// ---- POUs/20_AUTO/ST128/FB_AUT_128.TcPOU
FUNCTION_BLOCK FB_AUT_128 EXTENDS FB_AUT_ABSTRACT
(****************************************************************************)
(*	POU_AUT_zxx			Bausteinaufrufe Station	zxx							*)
(*	Status				ungetestet											*)
(*  Version:			1.0													*)
(*	Beschrieb:																*)
(*																			*)
(*	Abläufe:			FB_ABLzxxA		Hauptablauf							*)
(*																			*)
(*																			*)
(* 	25.09.2019/Dj															*)
(****************************************************************************)
(*	dd.mm.yyyy   KZ    x.y			Beschrieb								*)
(****************************************************************************)
VAR_INPUT
    (* spezifische Eingänge *)

END_VAR
VAR_OUTPUT
    (* spezifische Ausgänge *)

END_VAR
VAR
    (* Bausteine *)
    fb_TubeCapCheck : FB_ABL_128_TubeCapCheck; // 

    fb_stat : FB_AUT_Statistics;
END_VAR

(*******************************************************************)
(* Timer *)
(*******************************************************************)

(*******************************************************************)
(* Flanken / Merker *)
(*******************************************************************)
//MANU CYCLE
IF (enIN_State = StateMANU) AND xIN_ManuCycle THEN
    xManuCycle := TRUE;
END_IF;

IF (enIN_State <> StateMANU) OR xOUT_Done THEN
    xManuCycle := FALSE;
END_IF

//NEXT STEP
xNextStep := (enIN_State > StateSTEP) OR
             ((enIN_State = StateSTEP) AND xIN_Step) OR
             ((enIN_State = StateMANU) AND xManuCycle);

//RESET
xReset := (enIN_State < StateREADY) AND (enIN_State <> StateINIT) AND NOT xManuCycle;

(*******************************************************************)
(* Bausteinaufrufe Abläufe *)
(*******************************************************************)

xRelease := MAIN.MoverMan.IsProcessUsed(THIS^);

fb_TubeCapCheck(xIN_Reset       := xReset,
                xIN_Init        := xIN_Init,
                xIN_Quit        := xIN_Quit,
                xIN_Start       := enIN_State >= enState.StateLEER AND xRelease,
                xIN_Sperre      := NOT xIN_On,
                xIN_NextStep    := xNextStep,
                xIN_AlarmAktiv  := xIN_AlarmAktiv,
                xIN_DryCycle    := xIN_DryCycle,
                xIN_RestartCYCL := enIN_State >= enState.StateLEER,
                enIN_State      := enIN_State,
                tIN_Timeout     := tIN_Timeout,
                pxFG_Freigabe   := ADR(xRelease),
                Mover           := THIS^.Mover);

fb_stat(xIN_Enable  := enState.StateAUTO = enIN_State,
        xIN_Waiting := fb_TubeCapCheck.xOUT_Wait,
        xIN_Running := (fb_TubeCapCheck.iOUT_Step >= ST128_TubeCapCheck_e.START) AND
                       (fb_TubeCapCheck.iOUT_Step <= ST128_TubeCapCheck_e.DONE),
        // Since we use a mover system, a cycle is done when we are waiting on a mover
        xIN_Done := fb_TubeCapCheck.iOUT_Step = ST128_TubeCapCheck_e.waitOnMover);

(*******************************************************************)
(* Mover reset flags *)
(*******************************************************************)

(*******************************************************************)
(* OUTPUT *)
(*******************************************************************)
xOUT_InitDone := fb_TubeCapCheck.xOUT_InitDone;
xOUT_Ready    := fb_TubeCapCheck.xOUT_Ready;
xOUT_Done     := fb_TubeCapCheck.xOUT_Done;
xOUT_ErrFlag  := fb_TubeCapCheck.xOUT_ErrFlag;
xOUT_Wait     := fb_TubeCapCheck.xOUT_Wait;
xOUT_AlarmST  := xOUT_ErrFlag;

(*******************************************************************)
(* Bausteinaufruf Error Station *)
(*******************************************************************)
// POU_ERR_VORLAGE(xIN_QUIT:=xIN_Quit , pstrArIN_ALARM:=ADR(HMI.strArALARM[1]));

(* % of completion of the process *)
PROPERTY iCompletionPC : INT
GET
iCompletionPC := THIS^.fb_TubeCapCheck.iOUT_ProcessCompletion;
END_GET
END_PROPERTY

PROPERTY ProcessExecution : ProcessExecution_e
GET
ProcessExecution := THIS^._ProcessExecution;
END_GET
SET
THIS^._ProcessExecution := ProcessExecution;
END_SET
END_PROPERTY

PROPERTY xBusy : BOOL
GET
xBusy := THIS^.fb_TubeCapCheck.xOUT_Busy;
END_GET
SET
END_SET
END_PROPERTY

PROPERTY xDone : BOOL
GET
xDone := THIS^.fb_TubeCapCheck.xOUT_Ready OR THIS^.fb_TubeCapCheck.xOUT_Done;
END_GET
END_PROPERTY

PROPERTY xMoverPathFree : BOOL
GET
xMoverPathFree := THIS^.fb_TubeCapCheck.xOUT_MoverFree OR THIS^.fb_TubeCapCheck.xOUT_Ready OR THIS^.fb_TubeCapCheck.xOUT_Done;
END_GET
END_PROPERTY

PROPERTY xMoverShouldLeave : BOOL
GET
xMoverShouldLeave := THIS^.fb_TubeCapCheck.iOUT_Step = ST128_TubeCapCheck_e.SYNC_MOVER_LEAVE;
END_GET
END_PROPERTY

END_FUNCTION_BLOCK

// ---- POUs/20_AUTO/ST140/FB_AUT_140.TcPOU
FUNCTION_BLOCK FB_AUT_140 EXTENDS FB_AUT_ABSTRACT
(****************************************************************************)
(*	POU_AUT_zxx			Bausteinaufrufe Station	zxx							*)
(*	Status				ungetestet											*)
(*  Version:			1.0													*)
(*	Beschrieb:																*)
(*																			*)
(*	Abläufe:			FB_ABLzxxA		Hauptablauf							*)
(*																			*)
(*																			*)
(* 	25.09.2019/Dj															*)
(****************************************************************************)
(*	dd.mm.yyyy   KZ    x.y			Beschrieb								*)
(****************************************************************************)
VAR_INPUT
    (* spezifische Eingänge *)

END_VAR
VAR_OUTPUT
    (* spezifische Ausgänge *)

END_VAR
VAR
    (* Bausteine *)
    fb_Measure : FB_ABL_140_Measure;

    fb_stat : FB_AUT_Statistics;

END_VAR

(*******************************************************************)
(* Timer *)
(*******************************************************************)

(*******************************************************************)
(* Flanken / Merker *)
(*******************************************************************)
//MANU CYCLE
IF (enIN_State = StateMANU) AND xIN_ManuCycle THEN
    xManuCycle := TRUE;
END_IF;

IF (enIN_State <> StateMANU) OR xOUT_Done THEN
    xManuCycle := FALSE;
END_IF

//NEXT STEP
xNextStep := (enIN_State > StateSTEP) OR
             ((enIN_State = StateSTEP) AND xIN_Step) OR
             ((enIN_State = StateMANU) AND xManuCycle);

//RESET
xReset := (enIN_State < StateREADY) AND (enIN_State <> StateINIT) AND NOT xManuCycle;

(*******************************************************************)
(* Bausteinaufrufe Abläufe *)
(*******************************************************************)

xRelease := MAIN.MoverMan.IsProcessUsed(THIS^);

fb_Measure(xIN_Reset       := xReset,
           xIN_Init        := xIN_Init,
           xIN_Quit        := xIN_Quit,
           xIN_Start       := enIN_State >= enState.StateLEER AND xRelease,
           xIN_Sperre      := NOT xIN_On,
           xIN_NextStep    := xNextStep,
           xIN_AlarmAktiv  := xIN_AlarmAktiv,
           xIN_DryCycle    := xIN_DryCycle,
           xIN_RestartCYCL := enIN_State >= enState.StateLEER,
           enIN_State      := enIN_State,
           tIN_Timeout     := tIN_Timeout,
           pxFG_Freigabe   := ADR(xRelease),
           Mover           := THIS^.Mover);

fb_stat(xIN_Enable  := enState.StateAUTO = enIN_State,
        xIN_Waiting := fb_Measure.xOUT_Wait,
        xIN_Running := (fb_Measure.iOUT_Step >= ST140_Measure_e.START) AND
                       (fb_Measure.iOUT_Step <= ST140_Measure_e.DONE),
        // Since we use a mover system, a cycle is done when we are waiting on a mover
        xIN_Done := fb_Measure.iOUT_Step = ST140_Measure_e.waitOnMover);

(*******************************************************************)
(* Mover reset flags *)
(*******************************************************************)

(*******************************************************************)
(* OUTPUT *)
(*******************************************************************)
xOUT_InitDone := fb_Measure.xOUT_InitDone;
xOUT_Ready    := fb_Measure.xOUT_Ready;
xOUT_Done     := fb_Measure.xOUT_Done;
xOUT_ErrFlag  := fb_Measure.xOUT_ErrFlag;
xOUT_Wait     := fb_Measure.xOUT_Wait;
xOUT_AlarmST  := xOUT_ErrFlag;

(*******************************************************************)
(* Bausteinaufruf Error Station *)
(*******************************************************************)
// POU_ERR_VORLAGE(xIN_QUIT:=xIN_Quit , pstrArIN_ALARM:=ADR(HMI.strArALARM[1]));

(* % of completion of the process *)
PROPERTY iCompletionPC : INT
GET
iCompletionPC := THIS^.fb_Measure.iOUT_ProcessCompletion;
END_GET
END_PROPERTY

PROPERTY ProcessExecution : ProcessExecution_e
GET
ProcessExecution := THIS^._ProcessExecution;
END_GET
SET
THIS^._ProcessExecution := ProcessExecution;
END_SET
END_PROPERTY

PROPERTY xBusy : BOOL
GET
xBusy := THIS^.fb_Measure.xOUT_Busy;
END_GET
SET
END_SET
END_PROPERTY

PROPERTY xDone : BOOL
GET
xDone := THIS^.fb_Measure.xOUT_Ready OR THIS^.fb_Measure.xOUT_Done;
END_GET
END_PROPERTY

PROPERTY xMoverPathFree : BOOL
GET
xMoverPathFree := THIS^.fb_Measure.xOUT_MoverFree OR THIS^.fb_Measure.xOUT_Ready OR THIS^.fb_Measure.xOUT_Done;
END_GET
END_PROPERTY

PROPERTY xMoverShouldLeave : BOOL
GET
xMoverShouldLeave := THIS^.fb_Measure.iOUT_Step = ST140_Measure_e.SYNC_MOVER_LEAVE;
END_GET
END_PROPERTY

END_FUNCTION_BLOCK

// ---- POUs/20_AUTO/ST145/FB_AUT_145.TcPOU
FUNCTION_BLOCK FB_AUT_145 EXTENDS FB_AUT_ABSTRACT
(****************************************************************************)
(*	POU_AUT_zxx			Bausteinaufrufe Station	zxx							*)
(*	Status				ungetestet											*)
(*  Version:			1.0													*)
(*	Beschrieb:																*)
(*																			*)
(*	Abläufe:			FB_ABLzxxA		Hauptablauf							*)
(*																			*)
(*																			*)
(* 	25.09.2019/Dj															*)
(****************************************************************************)
(*	dd.mm.yyyy   KZ    x.y			Beschrieb								*)
(****************************************************************************)
VAR_INPUT
    (* spezifische Eingänge *)

END_VAR
VAR_OUTPUT
    (* spezifische Ausgänge *)

END_VAR
VAR
    (* Bausteine *)
    fb_Pnp    : FB_ABL_145_Pnp;
    fb_Feeder : FB_ABL_145_Feeder;

    fb_stat_pnp    : FB_AUT_Statistics;
    fb_stat_Feeder : FB_AUT_Statistics;

END_VAR

VAR CONSTANT
    ROT_TABLE_FREE_MAX_Y : REAL := 100.0; // If Y and Z axis is more than this value, the feeder cannot move
    ROT_TABLE_FREE_MAX_Z : REAL := 50.0; // If Z and Y axis is more than this value, the feeder cannot move

    PNP_VERTICAL_MAX_Z : REAL := 50.0; // If Z axis is more than this value, the horizontal axis of the pnp cannot move
END_VAR

(*******************************************************************)
(* Timer *)
(*******************************************************************)

(*******************************************************************)
(* Flanken / Merker *)
(*******************************************************************)
//MANU CYCLE
IF (enIN_State = StateMANU) AND xIN_ManuCycle THEN
    xManuCycle := TRUE;
END_IF;

IF (enIN_State <> StateMANU) OR xOUT_Done THEN
    xManuCycle := FALSE;
END_IF

//NEXT STEP
xNextStep := (enIN_State > StateSTEP) OR
             ((enIN_State = StateSTEP) AND xIN_Step) OR
             ((enIN_State = StateMANU) AND xManuCycle);

//RESET
xReset := (enIN_State < StateREADY) AND (enIN_State <> StateINIT) AND NOT xManuCycle;

(*******************************************************************)
(* Bausteinaufrufe Abläufe *)
(*******************************************************************)

xRelease := MAIN.MoverMan.IsProcessUsed(THIS^);

fb_Pnp(xIN_Reset          := xReset,
       xIN_Init           := xIN_Init,
       xIN_Quit           := xIN_Quit,
       xIN_Start          := enIN_State >= enState.StateLEER AND xRelease,
       xIN_Sperre         := NOT xIN_On,
       xIN_NextStep       := xNextStep,
       xIN_AlarmAktiv     := xIN_AlarmAktiv,
       xIN_DryCycle       := xIN_DryCycle,
       xIN_RestartCYCL    := enIN_State >= enState.StateLEER,
       enIN_State         := enIN_State,
       tIN_Timeout        := tIN_Timeout,
       pxFG_Freigabe      := ADR(xRelease),
       Mover              := THIS^.Mover,
       xIN_PceReadyToPick := fb_Feeder.xOUT_Done,
       xIN_HorAxisFree    := ST145_Axis.axis145_02Z.rActPos < ROT_TABLE_FREE_MAX_Y);

fb_Feeder(xIN_Reset       := xReset,
          xIN_Init        := xIN_Init,
          xIN_Quit        := xIN_Quit,
          xIN_Start       := enIN_State >= enState.StateLEER AND xRelease,
          xIN_Sperre      := NOT xIN_On,
          xIN_NextStep    := xNextStep,
          xIN_AlarmAktiv  := xIN_AlarmAktiv,
          xIN_DryCycle    := xIN_DryCycle,
          xIN_RestartCYCL := enIN_State >= enState.StateLEER,
          enIN_State      := enIN_State,
          tIN_Timeout     := tIN_Timeout,
          pxFG_Freigabe   := ADR(xRelease),
          // special
          xIN_PickPiece            := fb_Pnp.xOUT_PickPiece,
          xIN_RotTableBlockedByPnp := (ST145_Axis.axis145_01Y.rActPos > ROT_TABLE_FREE_MAX_Y) AND
                                      (ST145_Axis.axis145_02Z.rActPos > ROT_TABLE_FREE_MAX_Z));

fb_stat_pnp(xIN_Enable  := enState.StateAUTO = enIN_State,
            xIN_Waiting := fb_Pnp.xOUT_Wait,
            xIN_Running := (fb_Pnp.iOUT_Step >= ST145_Pnp_e.START) AND
                           (fb_Pnp.iOUT_Step <= ST145_Pnp_e.DONE),
            // Since we use a mover system, a cycle is done when we are waiting on a mover
            xIN_Done := fb_Pnp.iOUT_Step = ST145_Pnp_e.waitOnMover);

fb_stat_Feeder(xIN_Enable  := enState.StateAUTO = enIN_State,
               xIN_Waiting := fb_feeder.xOUT_Wait,
               xIN_Running := (fb_feeder.iOUT_Step >= ST145_Feeder_e.START) AND
                              (fb_feeder.iOUT_Step <= ST145_Feeder_e.DONE),
               xIN_Done := fb_feeder.iOUT_Step = ST145_Feeder_e.DONE);

(*******************************************************************)
(* Mover reset flags *)
(*******************************************************************)

(*******************************************************************)
(* OUTPUT *)
(*******************************************************************)
xOUT_InitDone := fb_Pnp.xOUT_InitDone AND fb_Feeder.xOUT_InitDone;
xOUT_Ready    := fb_Pnp.xOUT_Ready AND fb_Feeder.xOUT_Ready;
xOUT_Done     := fb_Pnp.xOUT_Done; // we ignore feeder
xOUT_ErrFlag  := fb_Pnp.xOUT_ErrFlag OR fb_Feeder.xOUT_ErrFlag;
xOUT_Wait     := fb_Pnp.xOUT_Wait AND fb_Feeder.xOUT_Wait;
xOUT_AlarmST  := xOUT_ErrFlag;

(*******************************************************************)
(* Bausteinaufruf Error Station *)
(*******************************************************************)
// POU_ERR_VORLAGE(xIN_QUIT:=xIN_Quit , pstrArIN_ALARM:=ADR(HMI.strArALARM[1]));

(* % of completion of the process *)
PROPERTY iCompletionPC : INT
GET
iCompletionPC := THIS^.fb_Pnp.iOUT_ProcessCompletion;
END_GET
END_PROPERTY

PROPERTY ProcessExecution : ProcessExecution_e
GET
ProcessExecution := THIS^._ProcessExecution;
END_GET
SET
THIS^._ProcessExecution := ProcessExecution;
END_SET
END_PROPERTY

PROPERTY xBusy : BOOL
GET
xBusy := THIS^.fb_Pnp.xOUT_Busy;
END_GET
SET
END_SET
END_PROPERTY

PROPERTY xDone : BOOL
GET
xDone := THIS^.fb_Pnp.xOUT_Ready OR THIS^.fb_Pnp.xOUT_Done;
END_GET
END_PROPERTY

PROPERTY xMoverPathFree : BOOL
GET
xMoverPathFree := THIS^.fb_Pnp.xOUT_MoverFree OR THIS^.fb_Pnp.xOUT_Ready OR THIS^.fb_Pnp.xOUT_Done;
END_GET
END_PROPERTY

PROPERTY xMoverShouldLeave : BOOL
GET
xMoverShouldLeave := THIS^.fb_Pnp.iOUT_Step = ST145_Pnp_e.SYNC_MOVER_LEAVE;
END_GET
END_PROPERTY

END_FUNCTION_BLOCK

// ---- POUs/20_AUTO/ST15x/FB_ABL_150.TcPOU
FUNCTION_BLOCK FB_ABL_150
(****************************************************************************************)
(*	TITEL				laden kristall- Modul	    										*)
(*	Status				ungetestet                         								*)
(*	Beschrieb:			Ablaufbeschreibung												*)
(*																						*)
(*	Steps:	self-explained using enum													*)
(***********************************Revisionen*******************************************)
(*	see github blames																	*)
(****************************************************************************************)

VAR_INPUT
    xIN_Reset       : BOOL;          // Schrittkette zurücksetzen 
    xIN_Init        : BOOL;          // Initialisieren
    xIN_Quit        : BOOL;          // Fehler quittieren 
    xIN_Start       : BOOL;          // Startbefehl
    xIN_Sperre      : BOOL;          // FB Sperren 
    xIN_NextStep    : BOOL;          // Nächsten Schritt ausführen 
    xIN_AlarmAktiv  : BOOL;          // Anlage hat Alarm
    xIN_DryCycle    : BOOL;          // Fahren ohne Teile
    xIN_RestartCYCL : BOOL;          // Zyklus erneut starten im STEP, END, LEERFAHREN
    enIN_State      : enState;       // Status Anlage
    tIN_Timeout     : TIME := T#10s; // Timout

    pxFG_Freigabe : POINTER TO BOOL; //Freigabe von Station

    // Application specific
    Mover : REFERENCE TO FB_Mover;

    xIN_capDetector             : BOOL;
    xIN_kraftubersetzunh_zuruck : BOOL;
    xIN_kraftubersetzunh_vor    : BOOL;
    pIN_ButtonMaintaining       : POINTER TO structButton;

    xIN_welding_bits : Ultrasonic_IN_bits_t;

    iIN_StationNumber : INT;    // station number 
    sIN_errorCodeSide : STRING; // added string to the error code, (e.g. left or right)

END_VAR
VAR_OUTPUT
    (* standart Ausgänge *)
    xOUT_ErrFlag  : BOOL;        // Error Flag 
    xOUT_Busy     : BOOL;        // Baustein befindet sich im Ablauf 
    xOUT_Done     : BOOL;        // Baustein hat den Ablauf beendet 		
    xOUT_Ready    : BOOL;        // Ready to begin, should be the same state as done	
    xOUT_Timeout  : BOOL;        // Timeout FB 
    xOUT_InitDone : BOOL;        // initialisierung fertig
    xOUT_Wait     : BOOL;        // Wartet auf Bedingung
    iOUT_Step     : ST150_Uss_e; // Aktueller Schritt 
    sOUT_Step     : STRING;      // Aktueller Schritt but in string format
    bOUT_Error    : BYTE;        // Fehlernummer

    iOUT_ProcessCompletion : INT;  //process completion, express in % (0-100)
    xOUT_MoverFree         : BOOL; // The mover is free to move

    xOUT_moverMaintening_valve : BOOL;
    xOUT_welding_bits          : Ultrasonic_OUT_bits_t;

END_VAR
VAR
    (* Standard *)
    (* Schritt *)
    iLastStep : ST150_Uss_e; // Merker letzter Schritt 
    iPreStep  : ST150_Uss_e; // Schritt zurück nach Alarm 
    iAktStep  : ST150_Uss_e; // aktueller Schritt

    // Trigger Starten 
    rtSTART : R_TRIG;
    // Timer TimeOut 
    TON_Timeout : TON;

    (* Bausteine *)

    (* Spezial *)
    fb_moverMaintening   : FB_ZylMo2El_V2_1;
    simu_moverMaintening : FB_Simu_Zyl2Pos;

    TON_UssError     : TON;
    TON_CapDetection : TON;

END_VAR
VAR CONSTANT
    USS_SIMULATION : BOOL := FALSE; // Set to TRUE to simulate this part of the program
END_VAR

(*******************************************************************)
(* Trigger  *)
(*******************************************************************)
(* Zurücksetzen *)
IF xIN_RESET THEN
    iPreStep  := ST150_Uss_e.RESET;
    iOUT_Step := ST150_Uss_e.RESET;
END_IF;

(* Error Quittieren *)
IF (bOUT_Error <> 0) AND xIN_Quit THEN
    xOUT_ErrFlag := FALSE;
    bOUT_Error   := 0;
    iOUT_Step    := iPreStep;
END_IF;

(*******************************************************************)
(* Timer *)
(*******************************************************************)
TON_Timeout(IN := xIN_NextStep AND (iLastStep = iOUT_Step) (*todo FG *) ,
            PT := tIN_Timeout);

TON_UssError(IN := ST150_Uss_e.uss_start = iOUT_Step,
             PT := DINT_TO_TIME(_20_AUTO.recipe.st150.USS_ErrorTime_ms));

TON_CapDetection(IN := ST150_Uss_e.check_cap_present = iOUT_Step,
                 PT := T#500MS);

(*******************************************************************)
(* Bausteine *)
(*******************************************************************)
fb_moverMaintening(xIN_Reset    := xIN_Reset OR (ST150_Uss_e.RESET = iOUT_Step),
                   xIN_Quit     := xIN_Quit,
                   xIN_Manu     := enState.StateMANU = enIN_State,
                   pbtIN_Button := pIN_ButtonMaintaining,
                   xIN_GS       := simu_moverMaintening.xOUT_inGS,
                   xIN_AS       := simu_moverMaintening.xOUT_inAS,
                   xIN_FREE     := TRUE,
                   xINtoGS      := (ST150_Uss_e.Init_ResetUss_maintaining_down = iOUT_Step) OR
                                   (ST150_Uss_e.mover_maintening_down = iOUT_Step),
                   xINtoAS   := ST150_Uss_e.mover_maintening_up = iOUT_Step,
                   tIN_ErrAS := DINT_TO_TIME(_20_AUTO.recipe.cylinder2Pos[StationList_e.ST150]
                                                 [ST150_Cylinders_e.Kraftbstutzung].toAS_alarm_time),
                   tIN_ErrGS := DINT_TO_TIME(_20_AUTO.recipe.cylinder2Pos[StationList_e.ST150]
                                                 [ST150_Cylinders_e.Kraftbstutzung].toGS_alarm_time),
                   tIN_WaitAS := DINT_TO_TIME(_20_AUTO.recipe.cylinder2Pos[StationList_e.ST150]
                                                  [ST150_Cylinders_e.Kraftbstutzung].toAS_wait_time),
                   tIN_WaitGS := DINT_TO_TIME(_20_AUTO.recipe.cylinder2Pos[StationList_e.ST150]
                                                  [ST150_Cylinders_e.Kraftbstutzung].toGS_wait_time));

simu_moverMaintening(xIN_Enable := USS_SIMULATION AND CONST.USE_SIMULATION,
                     xIN_inGS   := xIN_kraftubersetzunh_zuruck,
                     xIN_inAS   := xIN_kraftubersetzunh_vor,
                     xIN_valve  := fb_moverMaintening.xOUT_VALVE,
                     tIN_GS_ms  := 200,  // ms
                     tIN_AS_ms  := 200); // ms

(*******************************************************************)
(* OUTPUTS *)
(*******************************************************************)
// Error Flag 
xOUT_ErrFlag := (bOUT_Error <> 0) OR (ST150_Uss_e.ERROR = iOUT_Step);
// Baustein befindet sich im Ablauf 
xOUT_Busy := (iOUT_Step > ST150_Uss_e.READY) AND (iOUT_Step < ST150_Uss_e.DONE);
// Baustein hat den Ablauf beendet
xOUT_Done := (iOUT_Step = ST150_Uss_e.DONE);
// Process ready
xOUT_Ready := (iOUT_Step = ST150_Uss_e.READY) OR (iOUT_Step = ST150_Uss_e.waitOnMover);
// Timeout FB 				 		
xOUT_Timeout := TON_Timeout.Q;
// Itialisierung fertig			
xOUT_InitDone := (iOUT_Step = ST150_Uss_e.READY) OR (iOUT_Step = ST150_Uss_e.waitOnMover);
// Aktueller Schritt			
iOUT_Step := iOUT_Step; //Im Ablauf gesetzt		
sOUT_Step := TO_STRING(iOUT_Step);
//Fehlernummer	 
bOUT_Error := bOUT_Error; //Im Ablauf/FB gesetzt	
(* Warte (alle Schritte wo auf FG oder Teile gewartet wird) *)
xOUT_Wait := (iOUT_Step = ST150_Uss_e.DONE) OR
             (iOUT_Step = ST150_Uss_e.READY) OR
             (iOUT_Step = ST150_Uss_e.START) OR
             (iOUT_Step = ST150_Uss_e.waitOnMover) OR
             (iOUT_Step = ST150_Uss_e.SYNC_MOVER_LEAVE);

xOUT_MoverFree :=
    NOT (iOUT_Step >= ST150_Uss_e.MOVER_NEEDED_OP AND iOUT_Step < ST150_Uss_e.MOVER_FREE_OP) AND
    (iOUT_Step >= ST150_Uss_e.READY) AND
    (iOUT_Step < ST150_Uss_e.ERROR);

iOUT_ProcessCompletion := F_GetPercent_2(iAktStep,
                                         iAktStep,
                                         iAktStep,
                                         ST150_Uss_e.check_cap_present,
                                         ST150_Uss_e.SYNC_MOVER_LEAVE);

xOUT_moverMaintening_valve :=
    fb_moverMaintening.xOUT_VALVE AND NOT (USS_SIMULATION AND CONST.USE_SIMULATION);

xOUT_welding_bits.Start :=
    (ST150_Uss_e.uss_start = iOUT_Step) AND
    NOT (USS_SIMULATION AND CONST.USE_SIMULATION) AND
    xIN_capDetector;

xOUT_welding_bits.Reset :=
    (_14_STATE._FB_btQUIT.pbtIN^.press AND
    NOT (ST150_Uss_e.uss_working = iOUT_Step) AND
    NOT (ST150_Uss_e.uss_start = iOUT_Step)) OR
    (ST150_Uss_e.Init_ResetUss_maintaining_down = iOUT_Step);

xOUT_welding_bits.Data_Hex1 := _20_AUTO.recipe.st150.USS_Type.0; // _20_AUTO.recipe.st150.USS_Type = 1;
xOUT_welding_bits.Data_Hex2 := _20_AUTO.recipe.st150.USS_Type.1; // _20_AUTO.recipe.st150.USS_Type = 2;
xOUT_welding_bits.Data_Hex4 := _20_AUTO.recipe.st150.USS_Type.2; // _20_AUTO.recipe.st150.USS_Type = 3;
xOUT_welding_bits.Data_Hex8 := _20_AUTO.recipe.st150.USS_Type.3; // _20_AUTO.recipe.st150.USS_Type = 4;

(*******************************************************************)
(* Ablauf *)
(*******************************************************************)

(* Sperren *)
IF xIN_Sperre THEN
    iPreStep  := ST150_Uss_e.RESET;
    iOUT_Step := ST150_Uss_e.RESET;
    RETURN;
END_IF;

(* Schritt Merker *)
IF iAktStep <> iOUT_Step THEN
    iLastStep := iAktStep;
    iAktStep  := iOUT_Step;
END_IF

(* START *)
rtSTART(CLK := xIN_Start);

IF 0 = bOUT_Error THEN
    IF fb_moverMaintening.xOUT_ErrFlag THEN
        bOUT_Error := 11;
    ELSIF USS_SIMULATION AND CONST.USE_SIMULATION AND xIN_welding_bits.Fehler THEN
        bOUT_Error := 12;
    ELSIF TON_UssError.Q THEN
        bOUT_Error := 13;
    END_IF
ELSIF iOUT_Step < ST150_Uss_e.ERROR THEN
    iOUT_Step := ST150_Uss_e.ERROR;
END_IF

(*******************************************************************)
(* Schrittkette  *)
(*******************************************************************)
CASE iOUT_Step OF

(***** RESET *****)
ST150_Uss_e.RESET: (* Schritt 0-99 *)
    //Initialisierungen
    //Start Init Ablauf
    IF xIN_Init THEN
        iOUT_Step := ST150_Uss_e.INIT;
        //Start Manu Ablauf
    ELSIF enIN_State = StateMANU AND xIN_NextStep THEN
        iOUT_Step := ST150_Uss_e.INIT;
    END_IF;

(***** INIT *****)
ST150_Uss_e.INIT: (* Grundstellung ? *)
    iOUT_Step := ST150_Uss_e.Init_ResetUss_maintaining_down;

ST150_Uss_e.Init_ResetUss_maintaining_down:
    IF fb_moverMaintening.xOUT_inGS THEN
        iOUT_Step := ST150_Uss_e.READY;
    END_IF

(***** READY / INIT DONE *****)
ST150_Uss_e.READY:    (* Start AUTO,END,LEER,STEP *)
    IF xIN_Start THEN //IF rtSTART.Q THEN
        iOUT_Step := ST150_Uss_e.START;
    END_IF

(***** START  ZYKLISCH *****)
ST150_Uss_e.START: (*  *)
    IF xIN_NextStep AND pxFG_Freigabe^ THEN
        iOUT_Step := ST150_Uss_e.waitOnMover;
        iPreStep  := ST150_Uss_e.INIT;
    END_IF;

ST150_Uss_e.waitOnMover: (*  *)
    IF xIN_NextStep AND __ISVALIDREF(Mover) THEN
        IF Mover.GetLastStationDone() >= iIN_StationNumber THEN
            iOUT_Step := ST150_Uss_e.SYNC_MOVER_LEAVE;
        ELSIF Mover.GetLastStationDone() < INT#145 THEN
            iOUT_Step := ST150_Uss_e.SYNC_MOVER_LEAVE;
        ELSE
            iOUT_Step := ST150_Uss_e.check_cap_present;
            iPreStep  := ST150_Uss_e.waitOnMover;
        END_IF
    END_IF;

ST150_Uss_e.check_cap_present:
    IF xIN_capDetector OR (USS_SIMULATION AND CONST.USE_SIMULATION) THEN
        iOUT_Step := ST150_Uss_e.mover_maintening_up;
    ELSIF TON_CapDetection.Q THEN
        // Mover.SetErrorCode(CONCAT(CONCAT(INT_TO_STRING(iIN_StationNumber), '-B '), sIN_errorCodeSide));
        bOUT_Error := 8; // TODO to be removed
    END_IF

ST150_Uss_e.mover_maintening_up:
    IF xIN_NextStep AND fb_moverMaintening.xOUT_inAS THEN
        IF USS_SIMULATION AND CONST.USE_SIMULATION THEN
            iOUT_Step := ST150_Uss_e.mover_maintening_down;
        ELSE
            IF xIN_welding_bits.Bereit THEN
                iOUT_Step := ST150_Uss_e.uss_start;
                iPreStep  := ST150_Uss_e.waitOnMover;

                IF __ISVALIDREF(Mover) THEN
                    IF NOT Mover.SetLastStation(iIN_StationNumber) THEN
                        ASSERT(0);
                    END_IF
                END_IF
            ELSE
                // bOUT_Error := 1; // welding not ready
            END_IF
        END_IF;
    END_IF;

ST150_Uss_e.uss_start:
    IF xIN_NextStep AND NOT xIN_welding_bits.NullPosition THEN
        iOUT_Step := ST150_Uss_e.uss_working;
    END_IF

ST150_Uss_e.uss_working:
    IF xIN_NextStep AND
       (NOT xIN_welding_bits.US_on AND
       xIN_welding_bits.NullPosition) THEN
        iOUT_Step := ST150_Uss_e.mover_maintening_down;
    END_IF

ST150_Uss_e.mover_maintening_down:
    IF xIN_NextStep AND fb_moverMaintening.xOUT_inGS THEN
        iOUT_Step := ST150_Uss_e.SYNC_MOVER_LEAVE;

        IF __ISVALIDREF(Mover) THEN
            IF NOT Mover.SetLastStation(iIN_StationNumber) THEN
                ASSERT(0);
            END_IF
        END_IF
    END_IF;

ST150_Uss_e.SYNC_MOVER_LEAVE:
    // The mover needs to be taken by MoverMan
    IF NOT __ISVALIDREF(Mover) THEN
        iOUT_Step := ST150_Uss_e.DONE;
    END_IF

(***** DONE *****)
ST150_Uss_e.DONE: (* Letzter Schritt  *)
    IF NOT xIN_AlarmAktiv THEN
        //AUTO
        IF (enIN_State = StateAUTO) AND xIN_RestartCYCL THEN
            iOUT_Step := ST150_Uss_e.START;
            //STEP / END / LEERFAHREN restart
        ELSIF (enIN_State < StateAUTO) AND (enIN_State >= enState.StateSTEP) AND xIN_RestartCYCL THEN
            iOUT_Step := ST150_Uss_e.START;
            //STEP / END / LEERFAHREN fertig
        ELSIF (enIN_State = StateREADY) THEN
            iOUT_Step := ST150_Uss_e.READY;
        END_IF;
    END_IF;

(************ ERROR *************)
ST150_Uss_e.ERROR: (* ERROR *) ;

END_CASE;

END_FUNCTION_BLOCK

// ---- POUs/20_AUTO/ST15x/FB_ABL_150_solo.TcPOU
FUNCTION_BLOCK FB_ABL_150_solo
(****************************************************************************************)
(*	TITEL				laden kristall- Modul	    										*)
(*	Status				ungetestet                         								*)
(*	Beschrieb:			Ablaufbeschreibung												*)
(*																						*)
(*	Steps:	self-explained using enum													*)
(***********************************Revisionen*******************************************)
(*	see github blames																	*)
(****************************************************************************************)

VAR_INPUT
    xIN_Reset       : BOOL;          // Schrittkette zurücksetzen 
    xIN_Init        : BOOL;          // Initialisieren
    xIN_Quit        : BOOL;          // Fehler quittieren 
    xIN_Start       : BOOL;          // Startbefehl
    xIN_Sperre      : BOOL;          // FB Sperren 
    xIN_NextStep    : BOOL;          // Nächsten Schritt ausführen 
    xIN_AlarmAktiv  : BOOL;          // Anlage hat Alarm
    xIN_DryCycle    : BOOL;          // Fahren ohne Teile
    xIN_RestartCYCL : BOOL;          // Zyklus erneut starten im STEP, END, LEERFAHREN
    enIN_State      : enState;       // Status Anlage
    tIN_Timeout     : TIME := T#10s; // Timout

    pxFG_Freigabe : POINTER TO BOOL; //Freigabe von Station

    // Application specific
    Mover : REFERENCE TO FB_Mover;

    xIN_capDetector             : BOOL;
    xIN_kraftubersetzunh_zuruck : BOOL;
    xIN_kraftubersetzunh_vor    : BOOL;

    xIN_welding_bits : Ultrasonic_IN_bits_t;

    iIN_StationNumber : INT; // station number 

END_VAR
VAR_OUTPUT
    (* standart Ausgänge *)
    xOUT_ErrFlag  : BOOL;        // Error Flag 
    xOUT_Busy     : BOOL;        // Baustein befindet sich im Ablauf 
    xOUT_Done     : BOOL;        // Baustein hat den Ablauf beendet 		
    xOUT_Ready    : BOOL;        // Ready to begin, should be the same state as done	
    xOUT_Timeout  : BOOL;        // Timeout FB 
    xOUT_InitDone : BOOL;        // initialisierung fertig
    xOUT_Wait     : BOOL;        // Wartet auf Bedingung
    iOUT_Step     : ST150_Uss_e; // Aktueller Schritt 
    sOUT_Step     : STRING;      // Aktueller Schritt but in string format
    bOUT_Error    : BYTE;        // Fehlernummer

    iOUT_ProcessCompletion : INT;  //process completion, express in % (0-100)
    xOUT_MoverFree         : BOOL; // The mover is free to move

    xOUT_moverMaintening_valve : BOOL;
    xOUT_welding_bits          : Ultrasonic_OUT_bits_t;

END_VAR
VAR
    (* Standard *)
    (* Schritt *)
    iLastStep : ST150_Uss_e; // Merker letzter Schritt 
    iPreStep  : ST150_Uss_e; // Schritt zurück nach Alarm 
    iAktStep  : ST150_Uss_e; // aktueller Schritt

    // Trigger Starten 
    rtSTART : R_TRIG;
    // Timer TimeOut 
    TON_Timeout : TON;

    (* Bausteine *)

    (* Spezial *)
    fb_moverMaintening   : FB_ZylMo2El_V2_1;
    simu_moverMaintening : FB_Simu_Zyl2Pos;

    TON_UssError : TON;

    welding_right_done    : BOOL := FALSE;
    ton_wait_mover_in_pos : TON;

END_VAR
VAR CONSTANT
    USS_SIMULATION : BOOL := FALSE; // Set to TRUE to simulate this part of the program
END_VAR

(*******************************************************************)
(* Trigger  *)
(*******************************************************************)
(* Zurücksetzen *)
IF xIN_RESET THEN
    iPreStep  := ST150_Uss_e.RESET;
    iOUT_Step := ST150_Uss_e.RESET;
END_IF;

(* Error Quittieren *)
IF (bOUT_Error <> 0) AND xIN_Quit THEN
    xOUT_ErrFlag := FALSE;
    bOUT_Error   := 0;
    iOUT_Step    := ST150_Uss_e.INIT;
END_IF;

(*******************************************************************)
(* Timer *)
(*******************************************************************)
TON_Timeout(IN := xIN_NextStep AND (iLastStep = iOUT_Step) (*todo FG *) ,
            PT := tIN_Timeout);

TON_UssError(IN := ST150_Uss_e.uss_start = iOUT_Step,
             PT := DINT_TO_TIME(_20_AUTO.recipe.st150.USS_ErrorTime_ms));

ton_wait_mover_in_pos(IN := iOUT_Step = ST150_Uss_e.wait_shuttle_in_pos,
                      PT := T#1S);

(*******************************************************************)
(* Bausteine *)
(*******************************************************************)
fb_moverMaintening(xIN_Reset    := xIN_Reset OR (ST150_Uss_e.RESET = iOUT_Step),
                   xIN_Quit     := xIN_Quit,
                   xIN_Manu     := enState.StateMANU = enIN_State,
                   pbtIN_Button := ADR(HMI.btManuCylinders[StationList_e.ST150][1]),
                   xIN_GS       := simu_moverMaintening.xOUT_inGS,
                   xIN_AS       := simu_moverMaintening.xOUT_inAS,
                   xIN_FREE     := TRUE,
                   xINtoGS      := (ST150_Uss_e.Init_ResetUss_maintaining_down = iOUT_Step) OR
                                   (ST150_Uss_e.mover_maintening_down = iOUT_Step),
                   xINtoAS   := ST150_Uss_e.mover_maintening_up = iOUT_Step,
                   tIN_ErrAS := DINT_TO_TIME(_20_AUTO.recipe.cylinder2Pos[StationList_e.ST150]
                                                 [ST150_Cylinders_e.Kraftbstutzung].toAS_alarm_time),
                   tIN_ErrGS := DINT_TO_TIME(_20_AUTO.recipe.cylinder2Pos[StationList_e.ST150]
                                                 [ST150_Cylinders_e.Kraftbstutzung].toGS_alarm_time),
                   tIN_WaitAS := DINT_TO_TIME(_20_AUTO.recipe.cylinder2Pos[StationList_e.ST150]
                                                  [ST150_Cylinders_e.Kraftbstutzung].toAS_wait_time),
                   tIN_WaitGS := DINT_TO_TIME(_20_AUTO.recipe.cylinder2Pos[StationList_e.ST150]
                                                  [ST150_Cylinders_e.Kraftbstutzung].toGS_wait_time));

simu_moverMaintening(xIN_Enable := USS_SIMULATION AND CONST.USE_SIMULATION,
                     xIN_inGS   := xIN_kraftubersetzunh_zuruck,
                     xIN_inAS   := xIN_kraftubersetzunh_vor,
                     xIN_valve  := fb_moverMaintening.xOUT_VALVE,
                     tIN_GS_ms  := 200,  // ms
                     tIN_AS_ms  := 200); // ms

(*******************************************************************)
(* OUTPUTS *)
(*******************************************************************)
// Error Flag 
xOUT_ErrFlag := (bOUT_Error <> 0) OR (ST150_Uss_e.ERROR = iOUT_Step);
// Baustein befindet sich im Ablauf 
xOUT_Busy := (iOUT_Step > ST150_Uss_e.READY) AND (iOUT_Step < ST150_Uss_e.DONE);
// Baustein hat den Ablauf beendet
xOUT_Done := (iOUT_Step = ST150_Uss_e.DONE);
// Process ready
xOUT_Ready := (iOUT_Step = ST150_Uss_e.READY) OR (iOUT_Step = ST150_Uss_e.waitOnMover);
// Timeout FB 				 		
xOUT_Timeout := TON_Timeout.Q;
// Itialisierung fertig			
xOUT_InitDone := (iOUT_Step = ST150_Uss_e.READY) OR (iOUT_Step = ST150_Uss_e.waitOnMover);
// Aktueller Schritt			
iOUT_Step := iOUT_Step; //Im Ablauf gesetzt		
sOUT_Step := TO_STRING(iOUT_Step);
//Fehlernummer	 
bOUT_Error := bOUT_Error; //Im Ablauf/FB gesetzt	
(* Warte (alle Schritte wo auf FG oder Teile gewartet wird) *)
xOUT_Wait := (iOUT_Step = ST150_Uss_e.DONE) OR
             (iOUT_Step = ST150_Uss_e.READY) OR
             (iOUT_Step = ST150_Uss_e.START) OR
             (iOUT_Step = ST150_Uss_e.waitOnMover) OR
             (iOUT_Step = ST150_Uss_e.SYNC_MOVER_LEAVE);

xOUT_MoverFree :=
    NOT (iOUT_Step >= ST150_Uss_e.MOVER_NEEDED_OP AND iOUT_Step < ST150_Uss_e.MOVER_FREE_OP) AND
    (iOUT_Step >= ST150_Uss_e.READY) AND
    (iOUT_Step < ST150_Uss_e.ERROR);

iOUT_ProcessCompletion := F_GetPercent_2(iAktStep,
                                         iAktStep,
                                         iAktStep,
                                         ST150_Uss_e.check_cap_present,
                                         ST150_Uss_e.SYNC_MOVER_LEAVE);

xOUT_moverMaintening_valve :=
    fb_moverMaintening.xOUT_VALVE AND NOT (USS_SIMULATION AND CONST.USE_SIMULATION);

xOUT_welding_bits.Start :=
    (ST150_Uss_e.uss_start = iOUT_Step) AND
    NOT (USS_SIMULATION AND CONST.USE_SIMULATION) AND
    xIN_capDetector;

xOUT_welding_bits.Reset :=
    _14_STATE._FB_btQUIT.pbtIN^.press OR (ST150_Uss_e.Init_ResetUss_maintaining_down = iOUT_Step);

xOUT_welding_bits.Data_Hex1 := _20_AUTO.recipe.st150.USS_Type.0; // _20_AUTO.recipe.st150.USS_Type = 1;
xOUT_welding_bits.Data_Hex2 := _20_AUTO.recipe.st150.USS_Type.1; // _20_AUTO.recipe.st150.USS_Type = 2;
xOUT_welding_bits.Data_Hex4 := _20_AUTO.recipe.st150.USS_Type.2; // _20_AUTO.recipe.st150.USS_Type = 3;
xOUT_welding_bits.Data_Hex8 := _20_AUTO.recipe.st150.USS_Type.3; // _20_AUTO.recipe.st150.USS_Type = 4;

(*******************************************************************)
(* Ablauf *)
(*******************************************************************)

(* Sperren *)
IF xIN_Sperre THEN
    iPreStep  := ST150_Uss_e.RESET;
    iOUT_Step := ST150_Uss_e.RESET;
    RETURN;
END_IF;

(* Schritt Merker *)
IF iAktStep <> iOUT_Step THEN
    iLastStep := iAktStep;
    iAktStep  := iOUT_Step;
END_IF

(* START *)
rtSTART(CLK := xIN_Start);

IF 0 = bOUT_Error THEN
    IF fb_moverMaintening.xOUT_ErrFlag THEN
        bOUT_Error := 11;
    ELSIF USS_SIMULATION AND CONST.USE_SIMULATION AND xIN_welding_bits.Fehler THEN
        bOUT_Error := 12;
    ELSIF TON_UssError.Q THEN
        bOUT_Error := 13;
    END_IF
ELSIF iOUT_Step < ST150_Uss_e.ERROR THEN
    iOUT_Step := ST150_Uss_e.ERROR;
END_IF

(*******************************************************************)
(* Schrittkette  *)
(*******************************************************************)
CASE iOUT_Step OF

(***** RESET *****)
ST150_Uss_e.RESET: (* Schritt 0-99 *)
    //Initialisierungen
    //Start Init Ablauf
    IF xIN_Init THEN
        iOUT_Step := ST150_Uss_e.INIT;
        //Start Manu Ablauf
    ELSIF enIN_State = StateMANU AND xIN_NextStep THEN
        iOUT_Step := ST150_Uss_e.INIT;
    END_IF;

(***** INIT *****)
ST150_Uss_e.INIT: (* Grundstellung ? *)
    iOUT_Step := ST150_Uss_e.Init_ResetUss_maintaining_down;

ST150_Uss_e.Init_ResetUss_maintaining_down:
    IF fb_moverMaintening.xOUT_inGS THEN
        iOUT_Step := ST150_Uss_e.READY;
    END_IF

(***** READY / INIT DONE *****)
ST150_Uss_e.READY:    (* Start AUTO,END,LEER,STEP *)
    IF xIN_Start THEN //IF rtSTART.Q THEN
        iOUT_Step := ST150_Uss_e.START;
    END_IF

(***** START  ZYKLISCH *****)
ST150_Uss_e.START: (*  *)
    IF xIN_NextStep AND pxFG_Freigabe^ THEN
        iOUT_Step := ST150_Uss_e.waitOnMover;
    END_IF;

ST150_Uss_e.waitOnMover: (*  *)
    IF xIN_NextStep AND __ISVALIDREF(Mover) THEN
        IF Mover.GetLastStationDone() >= iIN_StationNumber THEN
            iOUT_Step := ST150_Uss_e.SYNC_MOVER_LEAVE;
        ELSE
            iOUT_Step := ST150_Uss_e.mover_maintening_up;
        END_IF
    END_IF;

ST150_Uss_e.check_cap_present:
    IF xIN_capDetector OR (USS_SIMULATION AND CONST.USE_SIMULATION) THEN
        iOUT_Step := ST150_Uss_e.mover_maintening_up;
    ELSE
        iOUT_Step := ST150_Uss_e.SYNC_MOVER_LEAVE;

        IF __ISVALIDREF(Mover) THEN
            IF NOT Mover.SetLastStation(-iIN_StationNumber) THEN
                ASSERT(0);
            END_IF
        END_IF
    END_IF

ST150_Uss_e.mover_maintening_up:
    IF xIN_NextStep AND fb_moverMaintening.xOUT_inAS THEN
        IF USS_SIMULATION AND CONST.USE_SIMULATION THEN
            iOUT_Step := ST150_Uss_e.mover_maintening_down;
        ELSE
            IF xIN_welding_bits.Bereit THEN
                iOUT_Step := ST150_Uss_e.uss_start;

                IF __ISVALIDREF(Mover) THEN
                    IF NOT Mover.SetLastStation(-150) THEN
                        ASSERT(0);
                    END_IF
                END_IF
            ELSE
                bOUT_Error := 1; // welding not ready
            END_IF
        END_IF;
    END_IF;

ST150_Uss_e.uss_start:
    IF xIN_NextStep AND NOT xIN_welding_bits.NullPosition THEN
        iOUT_Step := ST150_Uss_e.uss_working;
    END_IF

ST150_Uss_e.uss_working:
    IF xIN_NextStep AND
       (NOT xIN_welding_bits.US_on AND
       xIN_welding_bits.NullPosition) THEN
        iOUT_Step := ST150_Uss_e.mover_maintening_down;
    END_IF

ST150_Uss_e.mover_maintening_down:
    IF xIN_NextStep AND fb_moverMaintening.xOUT_inGS THEN
        iOUT_Step := ST150_Uss_e.move_shuttle_120_mm;
    END_IF;

ST150_Uss_e.move_shuttle_120_mm:
    IF xIN_NextStep AND __ISVALIDREF(Mover) AND_THEN Mover.MoveRelativeInsideStation(118.0) THEN
        iOUT_Step := ST150_Uss_e.wait_shuttle_in_pos;
    END_IF

ST150_Uss_e.wait_shuttle_in_pos:
    IF ton_wait_mover_in_pos.Q THEN
        IF welding_right_done THEN
            iOUT_Step          := ST150_Uss_e.SYNC_MOVER_LEAVE;
            welding_right_done := FALSE;

            IF __ISVALIDREF(Mover) THEN
                IF NOT Mover.SetLastStation(iIN_StationNumber) THEN
                    ASSERT(0);
                END_IF
            END_IF
        ELSE
            iOUT_Step          := ST150_Uss_e.check_cap_present;
            welding_right_done := TRUE;
        END_IF
    END_IF

ST150_Uss_e.SYNC_MOVER_LEAVE:
    // The mover needs to be taken by MoverMan
    IF NOT __ISVALIDREF(Mover) THEN
        iOUT_Step := ST150_Uss_e.DONE;
    END_IF

(***** DONE *****)
ST150_Uss_e.DONE: (* Letzter Schritt  *)
    IF NOT xIN_AlarmAktiv THEN
        //AUTO
        IF (enIN_State = StateAUTO) AND xIN_RestartCYCL THEN
            iOUT_Step := ST150_Uss_e.START;
            //STEP / END / LEERFAHREN restart
        ELSIF (enIN_State < StateAUTO) AND (enIN_State >= enState.StateSTEP) AND xIN_RestartCYCL THEN
            iOUT_Step := ST150_Uss_e.START;
            //STEP / END / LEERFAHREN fertig
        ELSIF (enIN_State = StateREADY) THEN
            iOUT_Step := ST150_Uss_e.READY;
        END_IF;
    END_IF;

(************ ERROR *************)
ST150_Uss_e.ERROR: (* ERROR *) ;

END_CASE;

END_FUNCTION_BLOCK

// ---- POUs/20_AUTO/ST16x/FB_ABL_160.TcPOU
FUNCTION_BLOCK FB_ABL_160
(****************************************************************************************)
(*	TITEL				laden kristall- Modul	    										*)
(*	Status				ungetestet                         								*)
(*	Beschrieb:			Ablaufbeschreibung												*)
(*																						*)
(*	Steps:	self-explained using enum													*)
(***********************************Revisionen*******************************************)
(*	see github blames																	*)
(****************************************************************************************)

VAR_INPUT
    xIN_Reset       : BOOL;          // Schrittkette zurücksetzen 
    xIN_Init        : BOOL;          // Initialisieren
    xIN_Quit        : BOOL;          // Fehler quittieren 
    xIN_Start       : BOOL;          // Startbefehl
    xIN_Sperre      : BOOL;          // FB Sperren 
    xIN_NextStep    : BOOL;          // Nächsten Schritt ausführen 
    xIN_AlarmAktiv  : BOOL;          // Anlage hat Alarm
    xIN_DryCycle    : BOOL;          // Fahren ohne Teile
    xIN_RestartCYCL : BOOL;          // Zyklus erneut starten im STEP, END, LEERFAHREN
    enIN_State      : enState;       // Status Anlage
    tIN_Timeout     : TIME := T#10s; // Timout

    pxFG_Freigabe : POINTER TO BOOL; //Freigabe von Station

    // Application specific
    Mover                  : REFERENCE TO FB_Mover;
    ref_fb_CETA            : REFERENCE TO FB_CETA_715;
    refAxis_01Z_beckhoff   : REFERENCE TO AxisBeckhoff_t; // reference of the axis GVL struct
    constAxis_01Z_Beckhoff : AxisLinMotConst_t;
    axis_01Z_LinearConfig  : LinearMotionMan_Config_t;
    iSelectedAxis          : Axis_e;
    axis_01Z_parIN_Buttons : POINTER TO ARRAY[0..8] OF structButton;
    refCylinderBp          : REFERENCE TO ARRAY[0..CONST.MAX_CYLINDER_PER_STATION] OF structButton;
    refCylinderConf        : REFERENCE TO ARRAY[0..CONST.MAX_CYLINDER_PER_STATION] OF Cylinder2Pos_config;

    // inputs
    uiIN_DisplacementSensorLeft  : UINT;
    uiIN_DisplacementSensorRight : UINT;
    IN_recipe                    : ST160_Recipe_t;
    iIN_StationNumber            : INT;

END_VAR
VAR_OUTPUT
    (* standart Ausgänge *)
    xOUT_ErrFlag  : BOOL;         // Error Flag 
    xOUT_Busy     : BOOL;         // Baustein befindet sich im Ablauf 
    xOUT_Done     : BOOL;         // Baustein hat den Ablauf beendet 		
    xOUT_Ready    : BOOL;         // Ready to begin, should be the same state as done	
    xOUT_Timeout  : BOOL;         // Timeout FB 
    xOUT_InitDone : BOOL;         // initialisierung fertig
    xOUT_Wait     : BOOL;         // Wartet auf Bedingung
    iOUT_Step     : ST160_CETA_e; // Aktueller Schritt 
    sOUT_Step     : STRING;       // Aktueller Schritt but in string format
    bOUT_Error    : BYTE;         // Fehlernummer

    iOUT_ProcessCompletion : INT;  //process completion, express in % (0-100)
    xOUT_MoverFree         : BOOL; // The mover is free to move

    // outputs
    xOUT_niederhalter_links         : BOOL;
    xOUT_niederhalter_rechts        : BOOL;
    xOUT_dichtung_pruflocker_links  : BOOL;
    xOUT_dichtung_pruflocker_rechts : BOOL;

END_VAR
VAR
    (* Standard *)
    (* Schritt *)
    iLastStep : ST160_CETA_e; // Merker letzter Schritt 
    iPreStep  : ST160_CETA_e; // Schritt zurück nach Alarm 
    iAktStep  : ST160_CETA_e; // aktueller Schritt

    // Trigger Starten 
    rtSTART : R_TRIG;
    // Timer TimeOut 
    TON_Timeout : TON;

    (* Bausteine *)
    fb_PnpVerAxis    : FB_LinearMotionMan;
    simu_axis160_01Z : FB_Simu_AxisLIN_V1_1;
    fb_axis160_01Z   : FB_AxisLIN_V1_1;

    (* Spezial *)
    fb_capMainteningLeft  : FB_ZylMo2El_V2_1;
    fb_capMainteningRight : FB_ZylMo2El_V2_1;

    simu_capMainteningLeft  : FB_Simu_Zyl2Pos;
    simu_capMainteningRight : FB_Simu_Zyl2Pos;

    fb_dichtung_left  : FB_ZylMo2El_V2_1;
    fb_dichtung_right : FB_ZylMo2El_V2_1;

    simu_dichtung_left  : FB_Simu_Zyl2Pos;
    simu_dichtung_right : FB_Simu_Zyl2Pos;

    xCETA_Result_OK : BOOL;
END_VAR

VAR_IN_OUT
    axisRef_Hardware   : AXIS_REF;
    axisRef_Simulation : AXIS_REF;
END_VAR

VAR CONSTANT
    CETA_SIMULATION : BOOL := FALSE; // Set to TRUE to simulate this part of the program
END_VAR

(*******************************************************************)
(* Trigger  *)
(*******************************************************************)
(* Zurücksetzen *)
IF xIN_RESET THEN
    iPreStep  := ST160_CETA_e.RESET;
    iOUT_Step := ST160_CETA_e.RESET;
END_IF;

(* Error Quittieren *)
IF (bOUT_Error <> 0) AND xIN_Quit THEN
    xOUT_ErrFlag := FALSE;
    bOUT_Error   := 0;
    iOUT_Step    := ST160_CETA_e.INIT;
END_IF;

(*******************************************************************)
(* Timer *)
(*******************************************************************)
TON_Timeout(IN := xIN_NextStep AND (iLastStep = iOUT_Step) (*todo FG *) ,
            PT := tIN_Timeout);

(*******************************************************************)
(* Bausteine *)
(*******************************************************************)
fb_PnpVerAxis(config          := axis_01Z_LinearConfig,
              xIN_Init        := enIN_State = enState.StateINIT,
              xIN_Reset       := xIN_Reset,
              lrIN_CurrPos    := fb_axis160_01Z.rOUT_ActPos,
              lrIN_Delta_mm   := 0.05,
              iIN_CurrentStep := iOUT_Step,
              iIN_moveNumber  := ST160_PnpVerPos_e._max);

simu_axis160_01Z(xIN_InSimu    := CETA_SIMULATION AND CONST.USE_SIMULATION,
                 rIN_PosActual := fb_axis160_01Z.rOUT_ActPos,
                 pIN_axisSimu  := ADR(axisRef_Simulation),
                 pIN_axisHW    := ADR(axisRef_Hardware),
                 rIN_PosMax    := constAxis_01Z_Beckhoff.POS_MAX,
                 rIN_PosMin    := constAxis_01Z_Beckhoff.POS_MIN,
                 rIN_PixMax    := 80,
                 rIN_PixMin    := 0);

fb_axis160_01Z(enIN_State       := enIN_State,
               parIN_Buttons    := axis_01Z_parIN_Buttons,
               xIN_DisButtons   :=,
               xIN_Quit         := xIN_Quit,
               xIN_AX5000       := TRUE,
               xIN_ENC_ABS      := TRUE, // TODO set accordingly
               xIN_PARAMok      := TRUE,
               xIN_FREE         := TRUE,
               xIN_FREE_HOME    := TRUE,
               rIN_POSMIN       := constAxis_01Z_Beckhoff.POS_MIN,
               rIN_POSMAX       := constAxis_01Z_Beckhoff.POS_MAX,
               rIN_VELOMAX      := constAxis_01Z_Beckhoff.VELO_MAX,
               rIN_VELOMANU     := constAxis_01Z_Beckhoff.VELO_MANU,
               rIN_VELOOPEN     := constAxis_01Z_Beckhoff.POS_MAX / 4,
               rIN_JogInc       := AXIS.rTeachIncAxis,
               rIN_VeloJogManu  := TO_REAL(AXIS.rJogVelo_pc),
               xIN_HomeExe      :=,
               xIN_HomeCalib    :=,
               xIN_Execute      := fb_PnpVerAxis.xOUT_Execute,
               xIN_HomeExe      :=,
               xIN_Relative     :=,
               rIN_Position     := TO_REAL(fb_PnpVerAxis.OUT_MoveProfile.lrPosition),
               rIN_Velocity     := TO_REAL(fb_PnpVerAxis.OUT_MoveProfile.lrVelocity),
               rIN_Acceleration := TO_REAL(fb_PnpVerAxis.OUT_MoveProfile.lrAccel),
               rIN_Deceleration := TO_REAL(fb_PnpVerAxis.OUT_MoveProfile.lrDecel),
               rIN_Jerk         := TO_REAL(fb_PnpVerAxis.OUT_MoveProfile.lrJerk),
               rIN_PosManu      := TO_REAL(axis_01Z_LinearConfig
                                               .movesList[AXIS.bTeachPos[iSelectedAxis]].lrPosition),
               xIN_Reset := (ST160_CETA_e.RESET = iOUT_Step) OR xIN_Reset,
               // output
               rOUT_ActPos => refAxis_01Z_beckhoff.rActPos,
               axisIN_REF  := simu_axis160_01Z.pOUT_axisRef^);

// pneumatics
fb_capMainteningLeft(xIN_Reset    := xIN_Reset OR (ST160_CETA_e.RESET = iOUT_Step),
                     xIN_Quit     := xIN_Quit,
                     xIN_Manu     := enState.StateMANU = enIN_State,
                     pbtIN_Button := ADR(refCylinderBp[1]),
                     xIN_GS       := simu_capMainteningLeft.xOUT_inGS,
                     xIN_AS       := simu_capMainteningLeft.xOUT_inAS,
                     xIN_FREE     := TRUE,
                     xINtoGS      := (ST160_CETA_e.Init_pneumatics = iOUT_Step) OR
                                     (ST160_CETA_e.handling_up = iOUT_Step),
                     xINtoAS   := IN_recipe.Use_element_left AND (ST160_CETA_e.handling_down = iOUT_Step),
                     tIN_ErrAS := DINT_TO_TIME(refCylinderConf
                                                   [ST160_Cylinders_e.Niederhalter_links].toAS_alarm_time),
                     tIN_ErrGS := DINT_TO_TIME(refCylinderConf
                                                   [ST160_Cylinders_e.Niederhalter_links].toGS_alarm_time),
                     tIN_WaitAS := DINT_TO_TIME(refCylinderConf
                                                    [ST160_Cylinders_e.Niederhalter_links].toAS_wait_time),
                     tIN_WaitGS := DINT_TO_TIME(refCylinderConf
                                                    [ST160_Cylinders_e.Niederhalter_links].toGS_wait_time));

simu_capMainteningLeft(xIN_Enable := TRUE, // CETA_SIMULATION AND CONST.USE_SIMULATION,
                       xIN_inGS   := UINT_TO_INT(uiIN_DisplacementSensorLeft) < 10,
                       xIN_inAS   := UINT_TO_INT(uiIN_DisplacementSensorLeft) > 200,
                       xIN_valve  := fb_capMainteningLeft.xOUT_VALVE,
                       tIN_GS_ms  := 200,  // ms
                       tIN_AS_ms  := 200); // ms

fb_capMainteningRight(xIN_Reset    := xIN_Reset OR (ST160_CETA_e.RESET = iOUT_Step),
                      xIN_Quit     := xIN_Quit,
                      xIN_Manu     := enState.StateMANU = enIN_State,
                      pbtIN_Button := ADR(refCylinderBp[2]),
                      xIN_GS       := simu_capMainteningRight.xOUT_inGS,
                      xIN_AS       := simu_capMainteningRight.xOUT_inAS,
                      xIN_FREE     := TRUE,
                      xINtoGS      := (ST160_CETA_e.Init_pneumatics = iOUT_Step) OR
                                      (ST160_CETA_e.handling_up = iOUT_Step),
                      xINtoAS := IN_recipe.Use_element_right AND (ST160_CETA_e.handling_down = iOUT_Step),
                      tIN_ErrAS
                          := DINT_TO_TIME(refCylinderConf
                                              [ST160_Cylinders_e.Niederhalter_rechts].toAS_alarm_time),
                      tIN_ErrGS := DINT_TO_TIME(refCylinderConf
                                                    [ST160_Cylinders_e.Niederhalter_rechts].toGS_alarm_time),
                      tIN_WaitAS := DINT_TO_TIME(refCylinderConf
                                                     [ST160_Cylinders_e.Niederhalter_rechts].toAS_wait_time),
                      tIN_WaitGS := DINT_TO_TIME(refCylinderConf
                                                     [ST160_Cylinders_e.Niederhalter_rechts].toGS_wait_time));

simu_capMainteningRight(xIN_Enable := TRUE, // CETA_SIMULATION AND CONST.USE_SIMULATION,
                        xIN_inGS   := UINT_TO_INT(uiIN_DisplacementSensorRight) < 10,
                        xIN_inAS   := UINT_TO_INT(uiIN_DisplacementSensorRight) > 200,
                        xIN_valve  := fb_capMainteningRight.xOUT_VALVE,
                        tIN_GS_ms  := 200,  // ms
                        tIN_AS_ms  := 200); // ms

fb_dichtung_left(xIN_Reset    := xIN_Reset OR (ST160_CETA_e.RESET = iOUT_Step),
                 xIN_Quit     := xIN_Quit,
                 xIN_Manu     := enState.StateMANU = enIN_State,
                 pbtIN_Button := ADR(refCylinderBp[3]),
                 xIN_GS       := simu_dichtung_left.xOUT_inGS,
                 xIN_AS       := simu_dichtung_left.xOUT_inAS,
                 xIN_FREE     := TRUE,
                 xINtoGS      := (ST160_CETA_e.Init_pneumatics = iOUT_Step) OR
                                 (ST160_CETA_e.unseal_piece = iOUT_Step),
                 xINtoAS   := IN_recipe.Use_element_left AND (ST160_CETA_e.seal_piece = iOUT_Step),
                 tIN_ErrAS := DINT_TO_TIME(refCylinderConf
                                               [ST160_Cylinders_e.Dichtung_prufglocke_links].toAS_alarm_time),
                 tIN_ErrGS := DINT_TO_TIME(refCylinderConf
                                               [ST160_Cylinders_e.Dichtung_prufglocke_links].toGS_alarm_time),
                 tIN_WaitAS := DINT_TO_TIME(refCylinderConf
                                                [ST160_Cylinders_e.Dichtung_prufglocke_links].toAS_wait_time),
                 tIN_WaitGS := DINT_TO_TIME(refCylinderConf
                                                [ST160_Cylinders_e.Dichtung_prufglocke_links].toGS_wait_time));

simu_dichtung_left(xIN_Enable := TRUE,                             // CETA_SIMULATION AND CONST.USE_SIMULATION,
                   xIN_inGS   := NOT fb_dichtung_right.xOUT_VALVE, // no sensor here
                   xIN_inAS   := fb_dichtung_right.xOUT_VALVE,     // no sensor here
                   xIN_valve  := fb_dichtung_left.xOUT_VALVE,
                   tIN_GS_ms  := 200,  // ms
                   tIN_AS_ms  := 200); // ms

fb_dichtung_right(xIN_Reset    := xIN_Reset OR (ST160_CETA_e.RESET = iOUT_Step),
                  xIN_Quit     := xIN_Quit,
                  xIN_Manu     := enState.StateMANU = enIN_State,
                  pbtIN_Button := ADR(refCylinderBp[4]),
                  xIN_GS       := simu_dichtung_right.xOUT_inGS,
                  xIN_AS       := simu_dichtung_right.xOUT_inAS,
                  xIN_FREE     := TRUE,
                  xINtoGS      := (ST160_CETA_e.Init_pneumatics = iOUT_Step) OR
                                  (ST160_CETA_e.unseal_piece = iOUT_Step),
                  xINtoAS   := IN_recipe.Use_element_right AND (ST160_CETA_e.seal_piece = iOUT_Step),
                  tIN_ErrAS := DINT_TO_TIME(refCylinderConf
                                                [ST160_Cylinders_e.Dichtung_prufglocke_rechts].toAS_alarm_time),
                  tIN_ErrGS := DINT_TO_TIME(refCylinderConf
                                                [ST160_Cylinders_e.Dichtung_prufglocke_rechts].toGS_alarm_time),
                  tIN_WaitAS := DINT_TO_TIME(refCylinderConf
                                                 [ST160_Cylinders_e.Dichtung_prufglocke_rechts].toAS_wait_time),
                  tIN_WaitGS := DINT_TO_TIME(refCylinderConf
                                                 [ST160_Cylinders_e.Dichtung_prufglocke_rechts].toGS_wait_time));

simu_dichtung_right(xIN_Enable := TRUE,                             // CETA_SIMULATION AND CONST.USE_SIMULATION,
                    xIN_inGS   := NOT fb_dichtung_right.xOUT_VALVE, // no sensor here
                    xIN_inAS   := fb_dichtung_right.xOUT_VALVE,     // no sensor here
                    xIN_valve  := fb_dichtung_right.xOUT_VALVE,
                    tIN_GS_ms  := 200,  // ms
                    tIN_AS_ms  := 200); // ms

(*******************************************************************)
(* OUTPUTS *)
(*******************************************************************)
// Error Flag 
xOUT_ErrFlag := (bOUT_Error <> 0) OR (ST160_CETA_e.ERROR = iOUT_Step);
// Baustein befindet sich im Ablauf 
xOUT_Busy := (iOUT_Step > ST160_CETA_e.READY) AND (iOUT_Step < ST160_CETA_e.DONE);
// Baustein hat den Ablauf beendet
xOUT_Done := (iOUT_Step = ST160_CETA_e.DONE);
// Process ready
xOUT_Ready := (iOUT_Step = ST160_CETA_e.READY) OR (iOUT_Step = ST160_CETA_e.waitOnMover);
// Timeout FB 				 		
xOUT_Timeout := TON_Timeout.Q;
// Itialisierung fertig			
xOUT_InitDone := (iOUT_Step = ST160_CETA_e.READY) OR (iOUT_Step = ST160_CETA_e.waitOnMover);
// Aktueller Schritt			
iOUT_Step := iOUT_Step; //Im Ablauf gesetzt		
sOUT_Step := TO_STRING(iOUT_Step);
//Fehlernummer	 
bOUT_Error := bOUT_Error; //Im Ablauf/FB gesetzt	
(* Warte (alle Schritte wo auf FG oder Teile gewartet wird) *)
xOUT_Wait := (iOUT_Step = ST160_CETA_e.DONE) OR
             (iOUT_Step = ST160_CETA_e.READY) OR
             (iOUT_Step = ST160_CETA_e.START) OR
             (iOUT_Step = ST160_CETA_e.waitOnMover) OR
             (iOUT_Step = ST160_CETA_e.SYNC_MOVER_LEAVE);

xOUT_MoverFree :=
    NOT (iOUT_Step >= ST160_CETA_e.MOVER_NEEDED_OP AND iOUT_Step < ST160_CETA_e.MOVER_FREE_OP) AND
    (iOUT_Step >= ST160_CETA_e.READY) AND
    (iOUT_Step < ST160_CETA_e.ERROR);

iOUT_ProcessCompletion := F_GetPercent_2(iAktStep,
                                         iAktStep,
                                         iAktStep,
                                         ST160_CETA_e.Init_pneumatics,
                                         ST160_CETA_e.SYNC_MOVER_LEAVE);

xOUT_niederhalter_links :=
    fb_capMainteningLeft.xOUT_VALVE AND NOT (CETA_SIMULATION AND CONST.USE_SIMULATION);

xOUT_niederhalter_rechts :=
    fb_capMainteningRight.xOUT_VALVE AND NOT (CETA_SIMULATION AND CONST.USE_SIMULATION);

xOUT_dichtung_pruflocker_links :=
    fb_dichtung_left.xOUT_VALVE AND NOT (CETA_SIMULATION AND CONST.USE_SIMULATION);

xOUT_dichtung_pruflocker_rechts :=
    fb_dichtung_right.xOUT_VALVE AND NOT (CETA_SIMULATION AND CONST.USE_SIMULATION);

(*******************************************************************)
(* Ablauf *)
(*******************************************************************)

(* Sperren *)
IF xIN_Sperre THEN
    iPreStep  := ST160_CETA_e.RESET;
    iOUT_Step := ST160_CETA_e.RESET;
    RETURN;
END_IF;

(* Schritt Merker *)
IF iAktStep <> iOUT_Step THEN
    iLastStep := iAktStep;
    iAktStep  := iOUT_Step;
END_IF

(* START *)
rtSTART(CLK := xIN_Start);

IF 0 = bOUT_Error THEN
    IF fb_axis160_01Z.xOUT_ErrFlag THEN
        bOUT_Error := 11;
    ELSIF fb_capMainteningLeft.xOUT_ErrFlag THEN
        bOUT_Error := 12;
    ELSIF fb_capMainteningRight.xOUT_ErrFlag THEN
        bOUT_Error := 13;
    END_IF
ELSIF iOUT_Step < ST160_CETA_e.ERROR THEN
    iOUT_Step := ST160_CETA_e.ERROR;
END_IF

(*******************************************************************)
(* Schrittkette  *)
(*******************************************************************)
CASE iOUT_Step OF

(***** RESET *****)
ST160_CETA_e.RESET: (* Schritt 0-99 *)
    //Initialisierungen
    //Start Init Ablauf
    IF xIN_Init THEN
        iOUT_Step := ST160_CETA_e.INIT;
        //Start Manu Ablauf
    ELSIF enIN_State = StateMANU AND xIN_NextStep THEN
        iOUT_Step := ST160_CETA_e.INIT;
    END_IF;

(***** INIT *****)
ST160_CETA_e.INIT: (* Grundstellung ? *)
    iOUT_Step := ST160_CETA_e.Init_pneumatics;

ST160_CETA_e.Init_pneumatics:
    IF (fb_capMainteningLeft.xOUT_inGS AND fb_capMainteningRight.xOUT_inGS) AND
       (fb_dichtung_left.xOUT_inGS AND fb_dichtung_right.xOUT_inGS) THEN
        iOUT_Step := ST160_CETA_e.Init_vertical_down;
    END_IF

ST160_CETA_e.Init_vertical_down:
    IF fb_PnpVerAxis.MoveTo(ST160_PnpVerPos_e.gs_down).xOUT_InPos THEN
        iOUT_Step := ST160_CETA_e.Init_set_program_number;
    END_IF

ST160_CETA_e.Init_set_program_number:
    IF ref_fb_CETA.SetProgramNumber(IN_recipe.Program_number) THEN
        iOUT_Step := ST160_CETA_e.READY;
    END_IF

(***** READY / INIT DONE *****)
ST160_CETA_e.READY:   (* Start AUTO,END,LEER,STEP *)
    IF xIN_Start THEN //IF rtSTART.Q THEN
        iOUT_Step := ST160_CETA_e.START;
    END_IF

(***** START  ZYKLISCH *****)
ST160_CETA_e.START: (*  *)
    IF xIN_NextStep AND pxFG_Freigabe^ THEN
        iOUT_Step       := ST160_CETA_e.waitOnMover;
        xCETA_Result_OK := FALSE;
    END_IF;

ST160_CETA_e.waitOnMover: (*  *)
    IF xIN_NextStep AND __ISVALIDREF(Mover) THEN
        IF (Mover.GetLastStationDone() >= iIN_StationNumber) OR Mover.IsPieceBad() THEN
            iOUT_Step := ST160_CETA_e.SYNC_MOVER_LEAVE;
        ELSIF Mover.GetLastStationDone() < INT#150 THEN
            iOUT_Step := ST160_CETA_e.SYNC_MOVER_LEAVE;
        ELSE
            iOUT_Step := ST160_CETA_e.handling_down;
        END_IF
    END_IF;

ST160_CETA_e.handling_down:
    IF (NOT IN_recipe.Use_element_left OR fb_capMainteningLeft.xOUT_inAS) AND
       (NOT IN_recipe.Use_element_right OR fb_capMainteningRight.xOUT_inAS) THEN
        iOUT_Step := ST160_CETA_e.vertical_up;
    END_IF

ST160_CETA_e.vertical_up:
    IF fb_PnpVerAxis.MoveTo(ST160_PnpVerPos_e.as_up).xOUT_InPos THEN
        iOUT_Step := ST160_CETA_e.seal_piece;
    END_IF

ST160_CETA_e.seal_piece:
    IF (NOT IN_recipe.Use_element_left OR fb_dichtung_left.xOUT_inAS) AND
       (NOT IN_recipe.Use_element_right OR fb_dichtung_right.xOUT_inAS) THEN
        IF CETA_SIMULATION AND CONST.USE_SIMULATION THEN
            iOUT_Step       := ST160_CETA_e.unseal_piece;
            xCETA_Result_OK := TRUE;
        ELSE
            iOUT_Step := ST160_CETA_e.CETA_start;
        END_IF
    END_IF

ST160_CETA_e.CETA_start:
    IF ref_fb_CETA.xOUT_ReadyToStart THEN
        IF ref_fb_CETA.StartMeasurement() THEN
            iOUT_Step := ST160_CETA_e.CETA_wait_on_result;
        ELSE
            bOUT_Error := 21;
        END_IF
    END_IF

ST160_CETA_e.CETA_wait_on_result:
    IF ref_fb_CETA.xOUT_DataReady THEN
        // this void call is needed to tell CETA function block
        // that we have read the result
        ref_fb_CETA.GetResult();
        iOUT_Step := ST160_CETA_e.unseal_piece;
    END_IF

ST160_CETA_e.unseal_piece:
    IF (NOT IN_recipe.Use_element_left OR fb_dichtung_left.xOUT_inGS) AND
       (NOT IN_recipe.Use_element_right OR fb_dichtung_right.xOUT_inGS) THEN
        iOUT_Step := ST160_CETA_e.vertical_down;
    END_IF

ST160_CETA_e.vertical_down:
    IF fb_PnpVerAxis.MoveTo(ST160_PnpVerPos_e.gs_down).xOUT_InPos THEN
        iOUT_Step := ST160_CETA_e.handling_up;
    END_IF

ST160_CETA_e.handling_up:
    IF fb_capMainteningLeft.xOUT_inGS AND fb_capMainteningRight.xOUT_inGS THEN
        iOUT_Step := ST160_CETA_e.SYNC_MOVER_LEAVE;
        iPreStep  := ST160_CETA_e.SYNC_MOVER_LEAVE;

        IF __ISVALIDREF(Mover) AND ref_fb_CETA.xOUT_Measure_1_GOOD AND ref_fb_CETA.xOUT_Measure_2_GOOD THEN
            IF NOT Mover.SetLastStation(iIN_StationNumber) THEN
                ASSERT(0);
            END_IF
        ELSIF __ISVALIDREF(Mover) THEN

            IF NOT ref_fb_CETA.xOUT_Measure_1_GOOD AND NOT ref_fb_CETA.xOUT_Measure_2_GOOD THEN
                Mover.SetErrorCode(CONCAT(INT_TO_STRING(iIN_StationNumber), '-C Both in error'));
				
            ELSIF NOT ref_fb_CETA.xOUT_Measure_1_GOOD THEN
                Mover.SetErrorCode(CONCAT(INT_TO_STRING(iIN_StationNumber), '-C Left'));
				
            ELSIF NOT ref_fb_CETA.xOUT_Measure_2_GOOD THEN
                Mover.SetErrorCode(CONCAT(INT_TO_STRING(iIN_StationNumber), '-C Right'));
				
            END_IF

            IF NOT Mover.SetLastStation(-iIN_StationNumber) THEN
                ASSERT(0);
            END_IF
        END_IF
    END_IF

ST160_CETA_e.SYNC_MOVER_LEAVE:
    // The mover needs to be taken by MoverMan
    IF NOT __ISVALIDREF(Mover) THEN
        iOUT_Step := ST160_CETA_e.DONE;
    END_IF

(***** DONE *****)
ST160_CETA_e.DONE: (* Letzter Schritt  *)
    IF NOT xIN_AlarmAktiv THEN
        //AUTO
        IF (enIN_State = StateAUTO) AND xIN_RestartCYCL THEN
            iOUT_Step := ST160_CETA_e.START;
            //STEP / END / LEERFAHREN restart
        ELSIF (enIN_State < StateAUTO) AND (enIN_State >= enState.StateSTEP) AND xIN_RestartCYCL THEN
            iOUT_Step := ST160_CETA_e.START;
            //STEP / END / LEERFAHREN fertig
        ELSIF (enIN_State = StateREADY) THEN
            iOUT_Step := ST160_CETA_e.READY;
        END_IF;
    END_IF;

(************ ERROR *************)
ST160_CETA_e.ERROR: (* ERROR *) ;

END_CASE;

END_FUNCTION_BLOCK

// ---- POUs/20_AUTO/ST175/Trumpf/FB_Laser_ABL.TcPOU
FUNCTION_BLOCK FB_Laser_ABL
VAR_INPUT
    xIN_Start          : BOOL;
    xIN_WarmUpLaser    : BOOL; // activate laser, only possible when cycle is not started
    sIN_FileName       : STRING := 'Someting here please';
    xIN_ResetData      : BOOL;                      // reset all data, used to ensure that the marking data are in the laser
    sIN_ErrorCode      : STRING(NUM_STRING_LENGTH); // error code to write when a station is in error
    xIN_StationInError : BOOL;                      // don't write normal data, write error data instead
END_VAR
VAR_OUTPUT
    xOUT_DONE  : BOOL;
    xOUT_ERROR : BOOL;
    xOUT_BUSY  : BOOL;
END_VAR
VAR
    iStep     : INT := 0;
    sDataTime : STRING(NUM_STRING_LENGTH);

    sLastName : STRING;                    // var used to see if last value has changed or not
    sLastNum  : STRING(NUM_STRING_LENGTH); // var used to see if last value has changed or not

    sReadableTime : STRING; // used to form a readable text

    fb_time : NT_GetTime;
END_VAR
VAR CONSTANT
    NUM_STRING_LENGTH : UDINT := 50; // maximum string length for the number
END_VAR

fb_time(NETID := '',
        START :=,
        TMOUT := T#1S);

IF xIN_ResetData THEN
    MEMSET(ADR(sLastName), 0, SIZEOF(sLastName));
    MEMSET(ADR(sLastNum), 0, SIZEOF(sLastNum));
END_IF

IF 0 = iStep AND xIN_WarmUpLaser AND if_SingleCmds.bReady THEN
    if_SingleCmds.iStepNr := 10; // TLV - Activate Laser / Open Shutter
    if_SingleCmds.bStart  := TRUE;
END_IF

CASE iStep OF

0: (* wait on start *)
    IF xIN_Start THEN
        iStep := 1000;
    END_IF

1000: (* TruMark *)
    IF if_SingleCmds.bReady THEN
        IF if_TruMark.Status.b6_LaserMalfunction THEN
            if_SingleCmds.iStepNr := 120; // TLV - Activate Laser / Open Shutter
            if_SingleCmds.bStart  := TRUE;
            iStep                 := 1010;
        ELSIF if_TruMark.Status.b0_Laser_On THEN
            iStep := 1040; // go to get the time
        ELSE
            iStep := 1020;
        END_IF;
    END_IF

1010: (* Reset Done*)
    IF if_SingleCmds.bReady THEN
        iStep := 1020;
    END_IF

1020: (* Laser ON *)
    IF if_SingleCmds.bReady THEN
        if_SingleCmds.iStepNr := 10; // TLV - Activate Laser / Open Shutter
        if_SingleCmds.bStart  := TRUE;
        iStep                 := 1030;
    END_IF;

1030: (* ON DONE*)
    IF if_SingleCmds.bReady THEN
        iStep := 1040;
    END_IF;

1040: (* get time *)
    fb_time.START := TRUE;
    iStep         := 1050;

1050: (* get time *)
    IF NOT fb_time.BUSY THEN
        fb_time.START := FALSE;
        iStep         := 1100;
    END_IF

1100: (* New FILE ? todo *)
    IF 0 = FIND(sLastName, sIN_FileName) OR (LEN(sLastName) <> LEN(sIN_FileName)) THEN
        iStep := 1110;
    ELSIF xIN_StationInError THEN
        iStep := 1110;
    ELSE
        iStep := 1130;
    END_IF

1110: (* Load File *)
    IF if_SingleCmds.bReady THEN
        if_SingleCmds.iStepNr     := 20; // TLV - Load Marking-File with 2 variables
        if_SingleCmds.sInputValue := CONCAT('C:\Aquis\', CONCAT(sIN_FileName, '.VLF'));
        sLastName                 := sIN_FileName;

        if_SingleCmds.bStart := TRUE;
        iStep                := 1120;
    END_IF

1120: (* Conversation *)
    IF if_SingleCmds.bReady THEN
        if_SingleCmds.iStepNr := 30; // TLV - Request state of conversion
        if_SingleCmds.bStart  := TRUE;
        iStep                 := 1130;
    END_IF

1130: (* New Var ? todo*)
    // date format : Y1M1D1D2M2Y2-Sx

    IF NOT xIN_StationInError THEN
        sDataTime[0] := F_ToASC(str := '0') + TO_BYTE((fb_time.TIMESTR.wYear MOD 100) / 10);  // Y1
        sDataTime[1] := F_ToASC(str := '0') + TO_BYTE((fb_time.TIMESTR.wMonth MOD 100) / 10); // M1
        sDataTime[2] := F_ToASC(str := '0') + TO_BYTE((fb_time.TIMESTR.wDay MOD 100) / 10);   // D1
        sDataTime[3] := F_ToASC(str := '0') + TO_BYTE(fb_time.TIMESTR.wDay MOD 10);           // D2
        sDataTime[4] := F_ToASC(str := '0') + TO_BYTE(fb_time.TIMESTR.wMonth MOD 10);         // M2
        sDataTime[5] := F_ToASC(str := '0') + TO_BYTE(fb_time.TIMESTR.wYear MOD 10);          // Y2
        sDataTime[6] := F_ToASC(str := '-');
        sDataTime[7] := F_ToASC(str := 'S');
        sDataTime[8] := F_ToASC(str := '1'); // TODO, team of the day
        sDataTime[9] := 0;
    ELSE
        sReadableTime := '';
        sReadableTime := CONCAT(CONCAT(sReadableTime, WORD_TO_STRING(fb_time.TIMESTR.wDay)), '.');
        sReadableTime := CONCAT(CONCAT(sReadableTime, WORD_TO_STRING(fb_time.TIMESTR.wMonth)), '.');
        sReadableTime := CONCAT(CONCAT(sReadableTime, WORD_TO_STRING(fb_time.TIMESTR.wYear)), ' ');
        sReadableTime := CONCAT(CONCAT(sReadableTime, WORD_TO_STRING(fb_time.TIMESTR.wHour)), 'h');
        sReadableTime := CONCAT(CONCAT(sReadableTime, WORD_TO_STRING(fb_time.TIMESTR.wMinute)), 'm');
        sReadableTime := CONCAT(CONCAT(sReadableTime, WORD_TO_STRING(fb_time.TIMESTR.wSecond)), 's');

        sDataTime := CONCAT(CONCAT(sIN_ErrorCode, '    '), sReadableTime);
    END_IF

    IF 0 = FIND(sLastNum, sDataTime) OR
       (LEN(sLastNum) <> LEN(sDataTime)) OR
       ((sDataTime[2] = F_ToASC(str := '0')) AND (sDataTime[3] = F_ToASC(str := '0'))) THEN
        iStep := 1140;
    ELSE
        iStep := 1170;
    END_IF

    MEMCPY(ADR(sLastNum), ADR(sDataTime), NUM_STRING_LENGTH);

1140: (* Set Var *)
    IF if_SingleCmds.bReady THEN
        if_SingleCmds.iStepNr := 35; // TLV - Set Variable
        // Variable name = 'Var1'	value = '3374'		Delimiter = ; --> will be replased with 0x00 in TruMark_Ethercat
        if_SingleCmds.sInputValue := CONCAT('Var1;', TO_STRING(sDataTime));

        if_SingleCmds.bStart := TRUE;
        iStep                := 1150;
    END_IF

1150: (* Var Done -> Convert *)
    IF if_SingleCmds.bReady THEN
        if_SingleCmds.iStepNr := 55; // TLV - Convert Marking File
        if_SingleCmds.bStart  := TRUE;
        iStep                 := 1160;
    END_IF

1160: (* Request Convert *)
    IF if_SingleCmds.bReady THEN
        if_SingleCmds.iStepNr := 30; // TLV - Request state of conversion
        if_SingleCmds.bStart  := TRUE;
        iStep                 := 1170;
    END_IF

1170: (* Request State *)
    IF if_SingleCmds.bReady THEN
        if_SingleCmds.iStepNr := 40; // TLV - Request Laser state
        if_SingleCmds.bStart  := TRUE;
        iStep                 := 1200;
    END_IF

1200: (* mark *)
    IF if_TruMark.Status.b0_Laser_On AND if_TruMark.Status.b1_Laser_Ready AND if_SingleCmds.bReady THEN
        if_SingleCmds.iStepNr := 50; // TLV - Activate Laser / Open Shutter
        if_SingleCmds.bStart  := TRUE;
        iStep                 := 1210;
    END_IF

// is done when safety signals are FALSE
// 1210: (* release laser *)
//     IF if_SingleCmds.bReady THEN
//         if_SingleCmds.iStepNr := 12; // TLV - Desactivate Laser
//         if_SingleCmds.bStart  := TRUE;
//         iStep                 := 1300;
//     END_IF

1210:
    IF if_TruMark.Status.b15_Mark_Active THEN
        iStep := 1220;
    END_IF

1220:
    IF NOT if_TruMark.Status.b15_Mark_Active THEN
        iStep := 1300;
    END_IF

1300: (* Check GS Datumsringüberwachung *)
    IF NOT xIN_Start THEN
        iStep := 0;
    END_IF

END_CASE

xOUT_DONE  := 1300 = iStep;
xOUT_BUSY  := (iStep >= 1000 AND iStep < 1300) OR NOT if_SingleCmds.bReady;
xOUT_ERROR := if_TruMark.bError;

END_FUNCTION_BLOCK

// ---- POUs/20_AUTO/Mover/VISU_MoverDetail.TcVIS
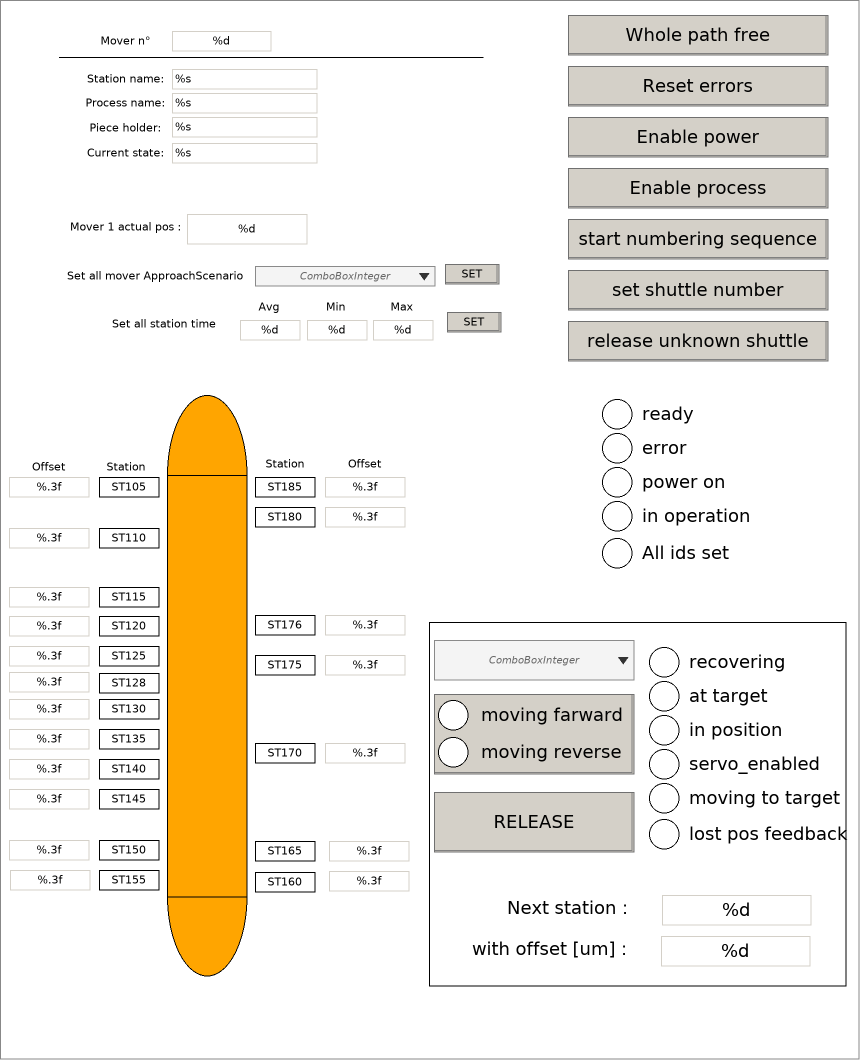
VISUALIZATION VISU_MoverDetail  // 860x1060
    Rectangle (429,622 417x364)
    Button (434,694 200x80)
        toggle gMoverAxis.Q_CT_Shuttle_to_BR.asStruct[HMI.selectedShuttle].bCommand.dirFarward
    Textfield (187,214 120x30), "%d", text variable: MAIN.MoverMan._MoverList[1]._MoverAxis._CurrentPos
        OnMouseDown: write the text variable via Default
    Label (38,212 146x30), "Mover 1 actual pos :"
    ComboBoxInteger (255,266 180x20), variable: MAIN.MoverMan.HMI_Scenario
    Label (59,261 187x30), "Set all mover ApproachScenario"
    Button (445,264 54x20), "SET"
        OnMouseDown: execute { MAIN.MoverMan.SetAllScenario(); }
    Label (93,309 126x30), "Set all station time"
    Textfield (240,320 60x20), "%d", text variable: MAIN.MoverMan.HMI_TimeAvg
        OnMouseDown: write the text variable via Default
    Label (241,296 56x22), "Avg"
    Textfield (307,320 60x20), "%d", text variable: MAIN.MoverMan.HMI_TimeMin
        OnMouseDown: write the text variable via Default
    Label (308,296 56x22), "Min"
    Textfield (373,320 60x20), "%d", text variable: MAIN.MoverMan.HMI_TimeMax
        OnMouseDown: write the text variable via Default
    Label (374,296 56x22), "Max"
    Button (447,312 54x20), "SET"
        OnMouseDown: execute { MAIN.MoverMan.SetAllTimers(ADR(PERS.iStationTimeDef1), 0); MAIN.MoverMan.SetAllTimers(ADR(PERS.iStationTimeDef2), 500); }
    Label (76,26 99x30), "Mover n°"
    Line (59,57) (483,57)
    Label (76,64 99x30), "Station name:"
    Label (76,88 99x30), "Process name:"
    Label (76,113 99x30), "Piece holder:"
    Label (76,138 99x30), "Current state:"
    Textfield (172,31 99x20), "%d", text variable: MAIN.MoverMan.HMI_iSelMover
        OnMouseDown: write the text variable via Default
    Textfield (172,69 145x20), "%s", text variable: MAIN.MoverMan._MoverList[MAIN.MoverMan.HMI_iSelMover].Station.ToString()
    Textfield (172,93 145x20), "%s"
    Textfield (172,117 145x20), "%s", text variable: MAIN.MoverMan._MoverList[MAIN.MoverMan.HMI_iSelMover].AttachedPieceHolder.ToString()
    Textfield (172,143 145x20), "%s", text variable: TO_STRING(MAIN.MoverMan._MoverList[MAIN.MoverMan.HMI_iSelMover]._State)
    Label (79,457 94x20), "Station"
    Label (-1,457 100x20), "Offset"
    Textfield (9,477 80x20), "%.3f", text variable: _20_AUTO.recipe.stationOffsets[StationList_e.ST105]
        OnMouseDown: write the text variable via Default
    Textfield (9,528 80x20), "%.3f", text variable: _20_AUTO.recipe.stationOffsets[StationList_e.ST110]
        OnMouseDown: write the text variable via Default
    Textfield (9,587 80x20), "%.3f", text variable: _20_AUTO.recipe.stationOffsets[StationList_e.ST115]
        OnMouseDown: write the text variable via Default
    Textfield (9,616 80x20), "%.3f", text variable: _20_AUTO.recipe.stationOffsets[StationList_e.ST120]
        OnMouseDown: write the text variable via Default
    Textfield (9,646 80x20), "%.3f", text variable: _20_AUTO.recipe.stationOffsets[StationList_e.ST125]
        OnMouseDown: write the text variable via Default
    Textfield (9,699 80x20), "%.3f", text variable: _20_AUTO.recipe.stationOffsets[StationList_e.ST130]
        OnMouseDown: write the text variable via Default
    Textfield (9,729 80x20), "%.3f", text variable: _20_AUTO.recipe.stationOffsets[StationList_e.ST135]
        OnMouseDown: write the text variable via Default
    Textfield (9,759 80x20), "%.3f", text variable: _20_AUTO.recipe.stationOffsets[StationList_e.ST140]
        OnMouseDown: write the text variable via Default
    Textfield (9,789 80x20), "%.3f", text variable: _20_AUTO.recipe.stationOffsets[StationList_e.ST145]
        OnMouseDown: write the text variable via Default
    Textfield (9,840 80x20), "%.3f", text variable: _20_AUTO.recipe.stationOffsets[StationList_e.ST150]
        OnMouseDown: write the text variable via Default
    Label (315,454 100x20), "Offset"
    Textfield (10,870 80x20), "%.3f", text variable: _20_AUTO.recipe.stationOffsets[StationList_e.ST155]
        OnMouseDown: write the text variable via Default
    Textfield (325,477 80x20), "%.3f", text variable: _20_AUTO.recipe.stationOffsets[StationList_e.ST185]
        OnMouseDown: write the text variable via Default
    Textfield (325,507 80x20), "%.3f", text variable: _20_AUTO.recipe.stationOffsets[StationList_e.ST180]
        OnMouseDown: write the text variable via Default
    Textfield (325,615 80x20), "%.3f", text variable: _20_AUTO.recipe.stationOffsets[StationList_e.ST176]
        OnMouseDown: write the text variable via Default
    Textfield (325,655 80x20), "%.3f", text variable: _20_AUTO.recipe.stationOffsets[StationList_e.ST175]
        OnMouseDown: write the text variable via Default
    Textfield (325,743 80x20), "%.3f", text variable: _20_AUTO.recipe.stationOffsets[StationList_e.ST170]
        OnMouseDown: write the text variable via Default
    Textfield (329,841 80x20), "%.3f", text variable: _20_AUTO.recipe.stationOffsets[StationList_e.ST165]
        OnMouseDown: write the text variable via Default
    Textfield (329,871 80x20), "%.3f", text variable: _20_AUTO.recipe.stationOffsets[StationList_e.ST160]
        OnMouseDown: write the text variable via Default
    Rectangle (99,870 60x20), "ST155", colour toggle: NOT GVL.st155_aut.xMoverPathFree
    Rectangle (99,840 60x20), "ST150", colour toggle: NOT GVL.st150_aut.xMoverPathFree
    Rectangle (99,789 60x20), "ST145", colour toggle: NOT GVL.st145_aut.xMoverPathFree
    Rectangle (99,759 60x20), "ST140", colour toggle: NOT GVL.st140_aut.xMoverPathFree
    Rectangle (99,729 60x20), "ST135", colour toggle: NOT GVL.st135_aut.xMoverPathFree
    Rectangle (99,699 60x20), "ST130", colour toggle: NOT GVL.st130_aut.xMoverPathFree
    Rectangle (99,646 60x20), "ST125", colour toggle: NOT GVL.st125_aut.xMoverPathFree
    Rectangle (99,616 60x20), "ST120", colour toggle: NOT GVL.st120_aut.xMoverPathFree
    Rectangle (99,587 60x20), "ST115", colour toggle: NOT GVL.st115_aut.xMoverPathFree
    Rectangle (99,528 60x20), "ST110", colour toggle: NOT GVL.st110_aut.xMoverPathFree
    Rectangle (99,477 60x20), "ST105", colour toggle: NOT GVL.st105_aut.xMoverPathFree
    Rectangle (255,507 60x20), "ST180", colour toggle: NOT GVL.st180_aut.xMoverPathFree
    Rectangle (255,615 60x20), "ST176", colour toggle: NOT GVL.st176_aut.xMoverPathFree
    Rectangle (255,655 60x20), "ST175", colour toggle: NOT GVL.st175_aut.xMoverPathFree
    Rectangle (255,743 60x20), "ST170", colour toggle: NOT GVL.st170_aut.xMoverPathFree
    Rectangle (255,841 60x20), "ST165", colour toggle: NOT GVL.st165_aut.xMoverPathFree
    Rectangle (255,872 60x20), "ST160", colour toggle: NOT GVL.st160_aut.xMoverPathFree
    Rectangle (255,477 60x20), "ST185", colour toggle: NOT GVL.st185_aut.xMoverPathFree
    Label (238,454 94x20), "Station"
    Ellipse (167,816 80x160)
    Ellipse (167,395 80x160)
    Rectangle (167,475 80x422)
    Button (568,66 260x40), "Reset errors", pressed state: gMoverAxis.Q_CT_Track_to_BR.asStruct.bCommand.resetErrors
    Button (568,117 260x40), "Enable power"
        toggle gMoverAxis.Q_CT_Track_to_BR.asStruct.bCommand.enablePower
    ComboBoxInteger (434,640 200x40), variable: HMI.selectedShuttle
    Button (434,792 200x60), "RELEASE", input disabled if: gMoverAxis.Q_CT_Track_to_BR.asStruct.bCommand.enableProcess OR NOT gMoverAxis.I_CT_Track_from_BR.asStruct.bStatus.allIdSet
        tap gMoverAxis.Q_CT_Shuttle_to_BR.asStruct[HMI.selectedShuttle].bCommand.release
    Ellipse (649,647 30x30), colour toggle: gMoverAxis.I_CT_Shuttle_from_BR.asStruct[HMI.selectedShuttle].bStatus.recovering
    Label (686,647 160x30), "recovering"
    Ellipse (649,681 30x30), colour toggle: gMoverAxis.I_CT_Shuttle_from_BR.asStruct[HMI.selectedShuttle].bStatus.at_target
    Label (686,681 160x30), "at target"
    Ellipse (649,715 30x30), colour toggle: gMoverAxis.I_CT_Shuttle_from_BR.asStruct[HMI.selectedShuttle].bStatus.in_position
    Label (686,715 160x30), "in position"
    Ellipse (649,749 30x30), colour toggle: gMoverAxis.I_CT_Shuttle_from_BR.asStruct[HMI.selectedShuttle].bStatus.servo_enabled
    Label (686,749 160x30), "servo_enabled"
    Ellipse (649,783 30x30), colour toggle: gMoverAxis.I_CT_Shuttle_from_BR.asStruct[HMI.selectedShuttle].bStatus.moving_to_load_target
    Label (686,783 160x30), "moving to target"
    Ellipse (649,819 30x30), colour toggle: gMoverAxis.I_CT_Shuttle_from_BR.asStruct[HMI.selectedShuttle].bStatus.lost_position_feedback
    Label (686,819 160x30), "lost pos feedback"
    Ellipse (602,399 30x30), colour toggle: gMoverAxis.I_CT_Track_from_BR.asStruct.bStatus.ready
    Label (639,399 160x30), "ready"
    Ellipse (602,433 30x30), colour toggle: gMoverAxis.I_CT_Track_from_BR.asStruct.bStatus.error
    Label (639,433 160x30), "error"
    Ellipse (602,467 30x30), colour toggle: gMoverAxis.I_CT_Track_from_BR.asStruct.bStatus.powerOn
    Label (639,467 160x30), "power on"
    Ellipse (602,501 30x30), colour toggle: gMoverAxis.I_CT_Track_from_BR.asStruct.bStatus.inOperation
    Label (639,501 160x30), "in operation"
    Button (568,168 260x40), "Enable process"
        toggle gMoverAxis.Q_CT_Track_to_BR.asStruct.bCommand.enableProcess
    Button (568,219 260x40), "start numbering sequence"
        toggle gMoverAxis.Q_CT_Track_to_BR.asStruct.bCommand.startMoverNumberingSequence
    Button (568,270 260x40), "set shuttle number"
        tap gMoverAxis.Q_CT_Track_to_BR.asStruct.bCommand.setShuttleNumber
    Button (568,321 260x40), "release unknown shuttle"
        tap gMoverAxis.Q_CT_Track_to_BR.asStruct.bCommand.releaseUnknownShuttle
    Ellipse (438,700 30x30), colour toggle: gMoverAxis.Q_CT_Shuttle_to_BR.asStruct[HMI.selectedShuttle].bCommand.dirFarward
    Ellipse (438,737 30x30), colour toggle: NOT gMoverAxis.Q_CT_Shuttle_to_BR.asStruct[HMI.selectedShuttle].bCommand.dirFarward
    Label (478,700 160x30), "moving farward"
    Label (478,737 160x30), "moving reverse"
    Button (568,15 260x40), "Whole path free"
        toggle gMoverAxis.Q_CT_Track_to_BR.asStruct.bCommand.wholePathFree
    Textfield (662,895 149x30), "%d", text variable: gMoverAxis.Q_CT_Shuttle_to_BR.asStruct[HMI.selectedShuttle].bNextStation
        OnMouseDown: write the text variable via Default
    Label (471,893 160x30), "Next station :"
    Textfield (661,936 149x30), "%d", text variable: gMoverAxis.Q_CT_Shuttle_to_BR.asStruct[HMI.selectedShuttle].diNextOffset_um
        OnMouseDown: write the text variable via Default
    Label (470,934 160x30), "with offset [um] :"
    Ellipse (602,538 30x30), colour toggle: gMoverAxis.I_CT_Track_from_BR.asStruct.bStatus.allIdSet
    Label (639,538 160x30), "All ids set"
    Textfield (9,672 80x20), "%.3f", text variable: _20_AUTO.recipe.stationOffsets[StationList_e.ST128]
        OnMouseDown: write the text variable via Default
    Rectangle (99,673 60x20), "ST128", colour toggle: NOT GVL.st125_aut.xMoverPathFree
END_VISUALIZATION

// ---- POUs/20_AUTO/ST115/VISU_Recipe_ST115.TcVIS
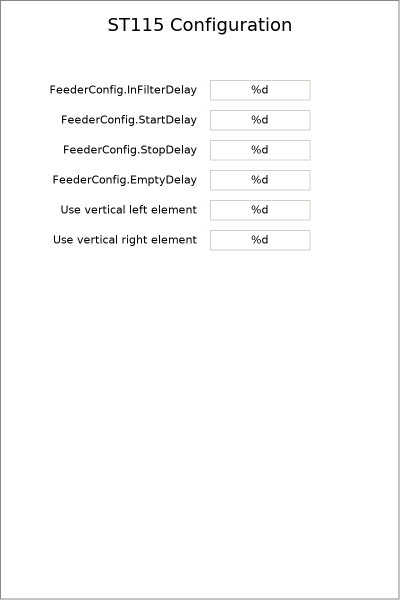
VISUALIZATION VISU_Recipe_ST115  // 400x600
    Textfield (210,80 100x20), "%d", text variable: _20_AUTO.recipe.st115.FeederConfig.InFilterDelay
        OnMouseDown: write the text variable via Default
    Label (0,5 400x40), "ST115 Configuration"
    Label (0,80 200x20), "FeederConfig.InFilterDelay"
    Textfield (210,110 100x20), "%d", text variable: _20_AUTO.recipe.st115.FeederConfig.StartDelay
        OnMouseDown: write the text variable via Default
    Label (0,110 200x20), "FeederConfig.StartDelay"
    Textfield (210,140 100x20), "%d", text variable: _20_AUTO.recipe.st115.FeederConfig.StopDelay
        OnMouseDown: write the text variable via Default
    Label (0,140 200x20), "FeederConfig.StopDelay"
    Textfield (210,170 100x20), "%d", text variable: _20_AUTO.recipe.st115.FeederConfig.EmptyDelay
        OnMouseDown: write the text variable via Default
    Label (0,170 200x20), "FeederConfig.EmptyDelay"
    Label (0,200 200x20), "Use vertical left element"
    Label (0,230 200x20), "Use vertical right element"
    Textfield (210,200 100x20), "%d", text variable: _20_AUTO.recipe.st115.xUseVerLeft
        OnMouseDown: write the text variable via Default
    Textfield (210,230 100x20), "%d", text variable: _20_AUTO.recipe.st115.xUseVerRight
        OnMouseDown: write the text variable via Default
END_VISUALIZATION

// ---- POUs/20_AUTO/ST115/VISU_ST115.TcVIS
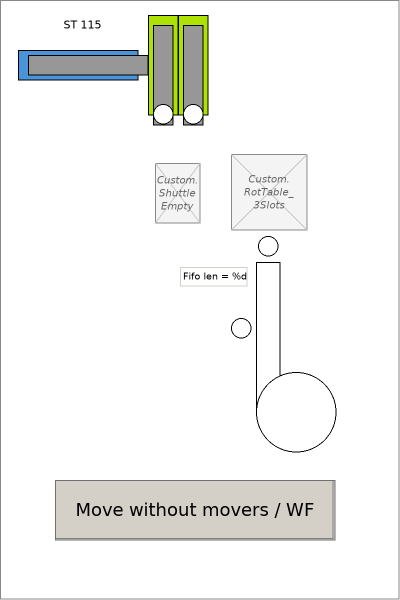
VISUALIZATION VISU_ST115  // 400x600
    Image (155,163 45x60), invisible if: NOT __ISVALIDREF(GVL.st115_aut._Mover), image: Custom.Shuttle Empty
    Image (231,154 76x76), image: Custom.RotTable_3Slots
        p2858320360: ST115_Axis.axis115_10W.rActPos
    Rectangle (18,50 120x30)
    Rectangle (28,55 120x20)
        p3560616238: GVL.st115_aut.fb_Pnp.fb_simu_axis115_01Y.rOUT_PixActual
    Rectangle (148,15 30x100)
        p3560616238: GVL.st115_aut.fb_Pnp.fb_simu_axis115_01Y.rOUT_PixActual
    Rectangle (153,25 20x100)
        p2738717112: GVL.st115_aut.fb_Pnp.fb_simu_axis115_02Z.rOUT_PixActual
        p3560616238: GVL.st115_aut.fb_Pnp.fb_simu_axis115_01Y.rOUT_PixActual
    Rectangle (178,15 30x100)
        p3560616238: GVL.st115_aut.fb_Pnp.fb_simu_axis115_01Y.rOUT_PixActual
    Rectangle (183,25 20x100)
        p2738717112: GVL.st115_aut.fb_Pnp.fb_simu_axis115_03Z.rOUT_PixActual
        p3560616238: GVL.st115_aut.fb_Pnp.fb_simu_axis115_01Y.rOUT_PixActual
    Rectangle (256,262 24x150)
    Ellipse (256,372 80x80), colour toggle: GVL.st115_aut.fb_Feeder.simu_feeder.xIN_Enable
    Ellipse (231,318 20x20), colour toggle: GVL.st115_aut.fb_Feeder.simu_feeder.xOUT_NewPiece
    Ellipse (153,104 20x20), colour toggle: GVL.st115_aut.fb_Pnp.fb_gripperLeft.xIN_AS
        p3560616238: GVL.st115_aut.fb_Pnp.fb_simu_axis115_01Y.rOUT_PixActual
        p2738717112: GVL.st115_aut.fb_Pnp.fb_simu_axis115_02Z.rOUT_PixActual
    Ellipse (183,104 20x20), colour toggle: GVL.st115_aut.fb_Pnp.fb_gripperRight.xIN_AS
        p2738717112: GVL.st115_aut.fb_Pnp.fb_simu_axis115_02Z.rOUT_PixActual
        p3560616238: GVL.st115_aut.fb_Pnp.fb_simu_axis115_01Y.rOUT_PixActual
    Ellipse (258,236 20x20), colour toggle: NOT GVL.st115_aut.fb_Feeder.simu_feeder.xOUT_NewPiece
    Textfield (180,267 67x19), "Fifo len = %d", text variable: GVL.st115_aut.fb_Feeder.simu_fifo_feeder_to_rotTable.GetLen()
    Label (40,15 85x20), "ST 115"
    Button (55,480 280x60), "Move without movers / WF", colour toggle: HMI.bArForceCyclusState[StationList_e.ST115]
        tap HMI.btArForceCyclus[StationList_e.ST115].button
END_VISUALIZATION

// ---- POUs/20_AUTO/ST120/VISU_ST120.TcVIS
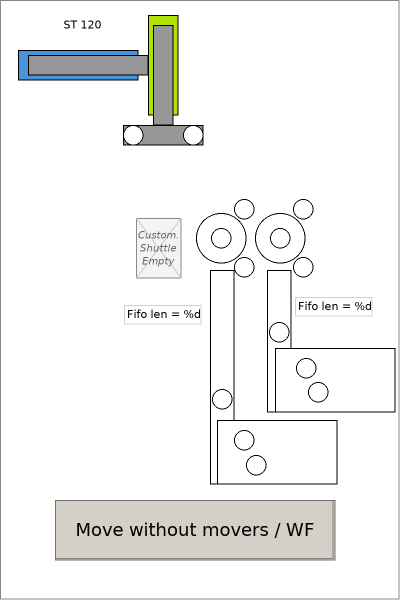
VISUALIZATION VISU_ST120  // 400x600
    Ellipse (196,213 50x50), colour toggle: GVL.st120_aut.fb_Feeder.fb_pivotLeft.xOUT_VALVE
    Image (136,218 45x60), invisible if: NOT __ISVALIDREF(GVL.st120_aut._Mover), image: Custom.Shuttle Empty
    Rectangle (18,50 120x30)
    Rectangle (28,55 120x20)
        p3560616238: GVL.st120_aut.fb_Pnp.fb_simu_axis120_01Y.rOUT_PixActual
    Rectangle (148,15 30x100)
        p3560616238: GVL.st120_aut.fb_Pnp.fb_simu_axis120_01Y.rOUT_PixActual
    Rectangle (153,25 20x100)
        p2738717112: GVL.st120_aut.fb_Pnp.fb_simu_axis120_02Z.rOUT_PixActual
        p3560616238: GVL.st120_aut.fb_Pnp.fb_simu_axis120_01Y.rOUT_PixActual
    Rectangle (210,270 24x214)
    Ellipse (212,389 20x20), colour toggle: GVL.st120_aut.fb_Feeder.simu_fifoLeft.IsFull()
    Ellipse (211,228 20x20), colour toggle: GVL.st120_aut.fb_Feeder.simu_fifoLeft.IsFull()
    Textfield (124,305 77x19), "Fifo len = %d", text variable: GVL.st120_aut.fb_Feeder.simu_fifoLeft.GetLen()
    Label (40,15 85x20), "ST 120"
    RoundedRectangle (217,420 120x64), colour toggle: GVL.st120_aut.fb_Feeder.fb_feederLeft.xOUT_EnableFeeder
    Rectangle (267,270 24x142)
    Ellipse (269,322 20x20), colour toggle: GVL.st120_aut.fb_Feeder.simu_fifoRight.IsFull()
    RoundedRectangle (275,348 120x64), colour toggle: GVL.st120_aut.fb_Feeder.fb_feederRight.xOUT_EnableFeeder
    Rectangle (123,125 80x20)
        p2738717112: GVL.st120_aut.fb_Pnp.fb_simu_axis120_02Z.rOUT_PixActual
        p3560616238: GVL.st120_aut.fb_Pnp.fb_simu_axis120_01Y.rOUT_PixActual
    Ellipse (183,125 20x20), colour toggle: GVL.st120_aut.fb_Pnp.fb_gripperRight.xIN_AS
        p3560616238: GVL.st120_aut.fb_Pnp.fb_simu_axis120_01Y.rOUT_PixActual
        p2738717112: GVL.st120_aut.fb_Pnp.fb_simu_axis120_02Z.rOUT_PixActual
    Ellipse (123,125 20x20), colour toggle: GVL.st120_aut.fb_Pnp.fb_gripperLeft.xIN_AS
        p3560616238: GVL.st120_aut.fb_Pnp.fb_simu_axis120_01Y.rOUT_PixActual
        p2738717112: GVL.st120_aut.fb_Pnp.fb_simu_axis120_02Z.rOUT_PixActual
    Textfield (295,297 77x19), "Fifo len = %d", text variable: GVL.st120_aut.fb_Feeder.simu_fifoRight.GetLen()
    Ellipse (255,213 50x50), colour toggle: GVL.st120_aut.fb_Feeder.fb_pivotRight.xOUT_VALVE
    Ellipse (270,228 20x20), colour toggle: GVL.st120_aut.fb_Feeder.simu_fifoRight.IsFull()
    Ellipse (293,199 20x20), colour toggle: GVL.st120_aut.fb_Feeder.fb_pivotRight.xIN_GS
    Ellipse (293,257 20x20), colour toggle: GVL.st120_aut.fb_Feeder.fb_pivotRight.xIN_AS
    Ellipse (234,199 20x20), colour toggle: GVL.st120_aut.fb_Feeder.fb_pivotLeft.xIN_GS
    Ellipse (234,257 20x20), colour toggle: GVL.st120_aut.fb_Feeder.fb_pivotLeft.xIN_AS
    Ellipse (246,455 20x20), colour toggle: GVL.st120_aut.fb_Feeder.fb_hubladerLeft.xIN_GS
    Ellipse (234,430 20x20), colour toggle: GVL.st120_aut.fb_Feeder.fb_hubladerLeft.xIN_AS
    Ellipse (296,358 20x20), colour toggle: GVL.st120_aut.fb_Feeder.fb_hubladerRight.xIN_AS
    Ellipse (308,382 20x20), colour toggle: GVL.st120_aut.fb_Feeder.fb_hubladerRight.xIN_GS
    Button (55,500 280x60), "Move without movers / WF", colour toggle: HMI.bArForceCyclusState[StationList_e.ST120]
        tap HMI.btArForceCyclus[StationList_e.ST120].button
END_VISUALIZATION

// ---- POUs/20_AUTO/ST125/VISU_ST125.TcVIS
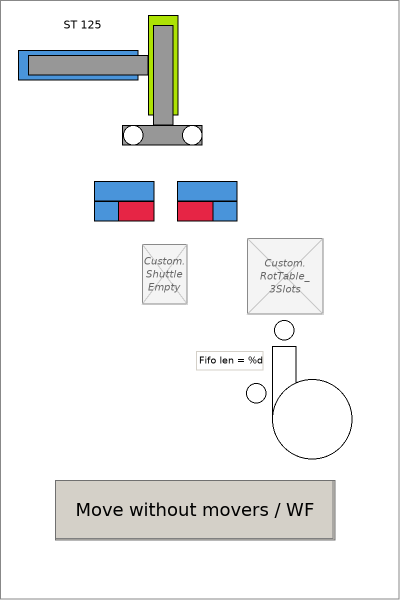
VISUALIZATION VISU_ST125  // 400x600
    Rectangle (187,201 50x20), invisible if: GVL.st125_aut.fb_Pnp.fb_handlingSolerohrRight.xIN_GS
    Rectangle (94,201 50x20), invisible if: GVL.st125_aut.fb_Pnp.fb_handlingSolerohrLeft.xIN_GS
    Rectangle (94,181 60x20), invisible if: GVL.st125_aut.fb_Pnp.fb_handlingSolerohrLeft.xIN_AS
    Rectangle (177,181 60x20), invisible if: GVL.st125_aut.fb_Pnp.fb_handlingSolerohrRight.xIN_AS
    Image (142,244 45x60), invisible if: NOT __ISVALIDREF(GVL.st125_aut._Mover), image: Custom.Shuttle Empty
    Image (247,238 76x76), image: Custom.RotTable_3Slots
        p2858320360: ST125_Axis.axis125_10W.rActPos
    Rectangle (18,50 120x30)
    Rectangle (28,55 120x20)
        p3560616238: GVL.st125_aut.fb_Pnp.fb_simu_axis125_01Y.rOUT_PixActual
    Rectangle (148,15 30x100)
        p3560616238: GVL.st125_aut.fb_Pnp.fb_simu_axis125_01Y.rOUT_PixActual
    Rectangle (153,25 20x100)
        p2738717112: GVL.st125_aut.fb_Pnp.fb_simu_axis125_02Z.rOUT_PixActual
        p3560616238: GVL.st125_aut.fb_Pnp.fb_simu_axis125_01Y.rOUT_PixActual
    Rectangle (272,346 24x73)
    Ellipse (272,379 80x80), colour toggle: GVL.st125_aut.fb_Feeder.simu_feeder.xIN_Enable
    Ellipse (246,383 20x20), colour toggle: GVL.st125_aut.fb_Feeder.simu_feeder.xOUT_NewPiece
    Ellipse (274,320 20x20)
    Textfield (196,351 67x19), "Fifo len = %d", text variable: GVL.st125_aut.fb_Feeder.simu_fifo_feeder_to_rotTable.GetLen()
    Label (40,15 85x20), "ST 125"
    Rectangle (122,125 80x20)
        p2738717112: GVL.st125_aut.fb_Pnp.fb_simu_axis125_02Z.rOUT_PixActual
        p3560616238: GVL.st125_aut.fb_Pnp.fb_simu_axis125_01Y.rOUT_PixActual
    Ellipse (123,125 20x20), colour toggle: GVL.st125_aut.fb_Pnp.fb_gripperFilterhutLeft.xIN_AS
        p3560616238: GVL.st125_aut.fb_Pnp.fb_simu_axis125_01Y.rOUT_PixActual
        p2738717112: GVL.st125_aut.fb_Pnp.fb_simu_axis125_02Z.rOUT_PixActual
    Ellipse (182,125 20x20), colour toggle: GVL.st125_aut.fb_Pnp.fb_gripperFilterhutRight.xIN_AS
        p3560616238: GVL.st125_aut.fb_Pnp.fb_simu_axis125_01Y.rOUT_PixActual
        p2738717112: GVL.st125_aut.fb_Pnp.fb_simu_axis125_02Z.rOUT_PixActual
    Rectangle (118,201 36x20), invisible if: NOT GVL.st125_aut.fb_Pnp.fb_gripperSolerohrLeft.xIN_AS
    Rectangle (177,201 36x20), invisible if: NOT GVL.st125_aut.fb_Pnp.fb_gripperSolerohrRight.xIN_AS
    Button (55,480 280x60), "Move without movers / WF", colour toggle: HMI.bArForceCyclusState[StationList_e.ST125]
        tap HMI.btArForceCyclus[StationList_e.ST125].button
END_VISUALIZATION

// ---- POUs/20_AUTO/ST128/VISU_Recipe_ST128.TcVIS
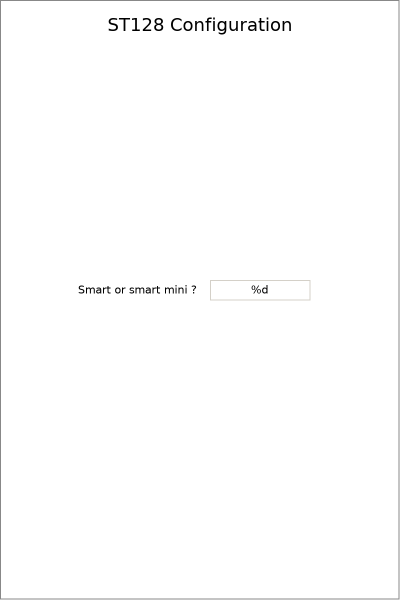
VISUALIZATION VISU_Recipe_ST128  // 400x600
    Label (0,5 400x40), "ST128 Configuration"
    Label (0,280 200x20), "Smart or smart mini ?"
    Textfield (210,280 100x20), "%d", text variable: _20_AUTO.recipe.st128.xIsTypeMiniOrSmart
        OnMouseDown: write the text variable via Default
END_VISUALIZATION

// ---- POUs/20_AUTO/ST140/VISU_Recipe_ST140.TcVIS
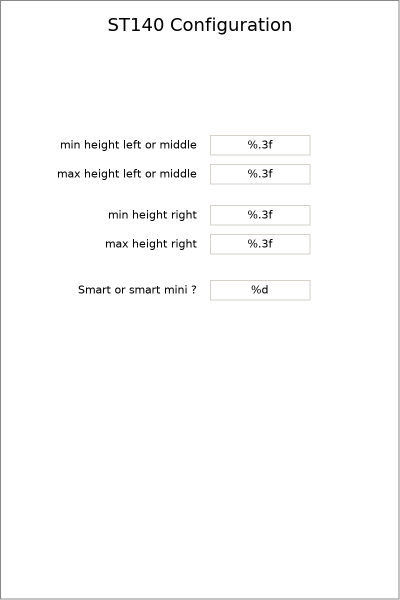
VISUALIZATION VISU_Recipe_ST140  // 400x600
    Label (0,5 400x40), "ST140 Configuration"
    Label (0,280 200x20), "Smart or smart mini ?"
    Textfield (210,280 100x20), "%d", text variable: _20_AUTO.recipe.st140.xIsTypeMiniOrSmart
        OnMouseDown: write the text variable via Default
    Label (0,135 200x20), "min height left or middle"
    Textfield (210,135 100x20), "%.3f", text variable: _20_AUTO.recipe.st140.rMinHeightSensorLeft
        OnMouseDown: write the text variable via Default
    Label (0,164 200x20), "max height left or middle"
    Textfield (210,164 100x20), "%.3f", text variable: _20_AUTO.recipe.st140.rMaxHeightSensorLeft
        OnMouseDown: write the text variable via Default
    Label (0,205 200x20), "min height right"
    Textfield (210,205 100x20), "%.3f", text variable: _20_AUTO.recipe.st140.rMinHeightSensorRight
        OnMouseDown: write the text variable via Default
    Label (0,234 200x20), "max height right"
    Textfield (210,234 100x20), "%.3f", text variable: _20_AUTO.recipe.st140.rMaxHeightSensorRight
        OnMouseDown: write the text variable via Default
END_VISUALIZATION

// ---- POUs/20_AUTO/ST16x/VISU_Recipe_ST160.TcVIS
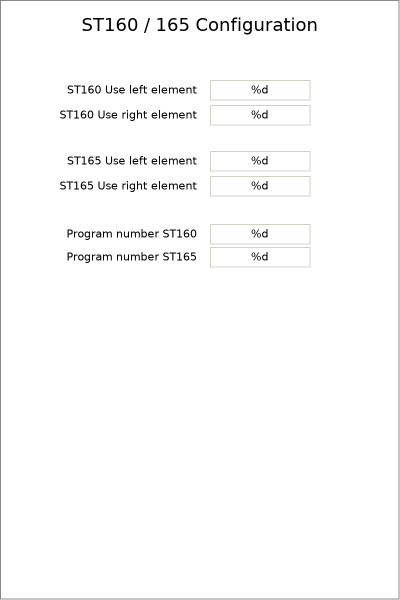
VISUALIZATION VISU_Recipe_ST160  // 400x600
    Textfield (210,80 100x20), "%d", text variable: _20_AUTO.recipe.st160.Use_element_left
        OnMouseDown: write the text variable via Default
    Label (0,5 400x40), "ST160 / 165 Configuration"
    Label (0,80 200x20), "ST160 Use left element"
    Textfield (210,105 100x20), "%d", text variable: _20_AUTO.recipe.st160.Use_element_right
        OnMouseDown: write the text variable via Default
    Label (0,105 200x20), "ST160 Use right element"
    Textfield (210,151 100x20), "%d", text variable: _20_AUTO.recipe.st165.Use_element_left
        OnMouseDown: write the text variable via Default
    Label (0,151 200x20), "ST165 Use left element"
    Textfield (210,176 100x20), "%d", text variable: _20_AUTO.recipe.st165.Use_element_right
        OnMouseDown: write the text variable via Default
    Label (0,176 200x20), "ST165 Use right element"
    Textfield (210,224 100x20), "%d", text variable: _20_AUTO.recipe.st160.Program_number
        OnMouseDown: write the text variable via Default
    Label (0,224 200x20), "Program number ST160"
    Textfield (210,247 100x20), "%d", text variable: _20_AUTO.recipe.st165.Program_number
        OnMouseDown: write the text variable via Default
    Label (0,247 200x20), "Program number ST165"
END_VISUALIZATION

// ---- POUs/20_AUTO/ST175/VISU_Recipe_ST175.TcVIS
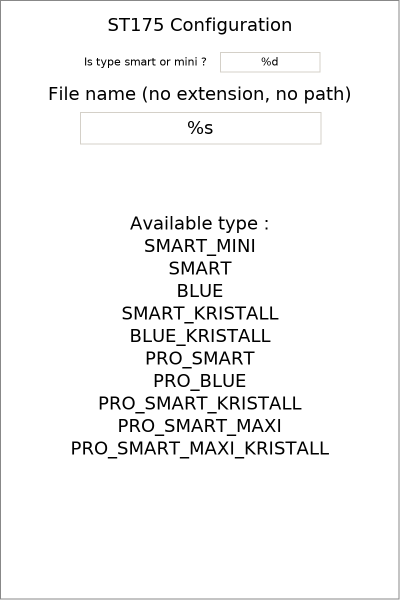
VISUALIZATION VISU_Recipe_ST175  // 400x600
    Textfield (80,112 241x32), "%s", text variable: _20_AUTO.recipe.st175.file_name
        OnMouseDown: write the text variable via Default
    Label (0,5 400x40), "ST175 Configuration"
    Label (24,84 352x20), "File name (no extension, no path)"
    Label (59,174 282x324), "Available type : SMART_MINI SMART BLUE SMART_KRISTALL BLUE_KRISTALL PRO_SMART PRO_BLUE PRO_SMART_KRISTALL PRO_SMART_MAXI PRO_SMART_MAXI_KRISTALL"
    Textfield (220,52 100x20), "%d", text variable: _20_AUTO.recipe.st175.isTypeSmartOrMini
        OnMouseDown: write the text variable via Default
    Label (10,52 200x20), "Is type smart or mini ?"
END_VISUALIZATION

// ---- POUs/20_AUTO/ST175/VISU_ST175.TcVIS
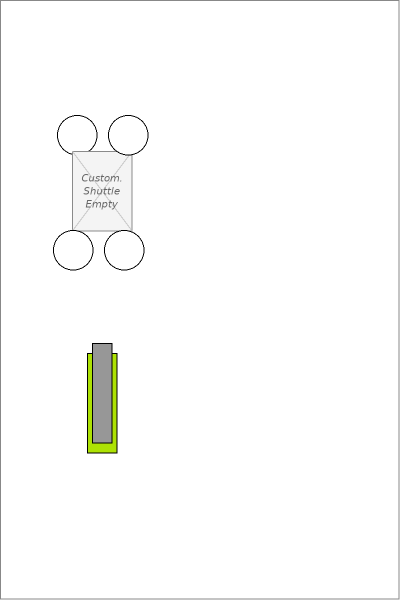
VISUALIZATION VISU_ST175  // 400x600
    Ellipse (57,115 40x40), colour toggle: GVL.st160_aut.fb_ABL_CETA.fb_capMainteningLeft.xIN_AS
    Image (72,151 60x80), angle 90, invisible if: NOT __ISVALIDREF(GVL.st160_aut._Mover), image: Custom.Shuttle Empty
    Ellipse (108,115 40x40), colour toggle: GVL.st160_aut.fb_ABL_CETA.fb_capMainteningRight.xIN_AS
    Rectangle (87,353 30x100)
    Rectangle (92,343 20x100)
        p2738717112: -GVL.st160_aut.fb_ABL_CETA.simu_axis160_01Z.rOUT_PixActual
    Ellipse (53,230 40x40), colour toggle: GVL.st160_aut.fb_ABL_CETA.fb_dichtung_left.xIN_AS
    Ellipse (104,230 40x40), colour toggle: GVL.st160_aut.fb_ABL_CETA.fb_dichtung_right.xIN_AS
END_VISUALIZATION

